ABB RAPID module: GoFa_GeneratedModule.modx

Module ACADIA_WORKSHOP_00_TEST
!Declarations

!jointtarget
VAR jointtarget TGofa_InitialConfig:=[[0,0,0,0,90,0],[9E9,9E9,9E9,9E9,9E9,9E9]];

!robtarget (Not Used for MoveAbsJ)
!VAR robtarget TGofa_0_End:=[[365,77.458,68.392],[0.707107,0,0,0.707107],[-1,0,0,0],[9E9,9E9,9E9,9E9,9E9,9E9]];

!speeddata (mm/s for the TCP, degrees/s for reorientation of the tool, mm/s for linear external axes, degrees/s for rotating external axes)
VAR speeddata speeddata0:=[200,80,5000,1000];

!tooldata (Not Used)
!PERS tooldata PonGoFa:=[True,[[-36.666,0.002,138.175],[0,0.92388,0,0.382683]],[0.001,[0,0,0.1],[1,0,0,0],0,0,0]];

!wobjdata (Not Used for MoveAbsJ)
!PERS wobjdata Root:=[False,True,"",[[0,0,0],[1,0,0,0]],[[0,0,0],[1,0,0,0]]];

!zonedata (Blend)
VAR zonedata DefaultBlend:=[False,1,0.1,1,0.1,1,0.1];
VAR zonedata FinePoint:=[True,1,0.1,1,0.1,1,0.1];

Proc Main()
  !Path Acceleration Limitation, units is m/s2, syntax: PathAccLim AccLim [\AccMax] DecelLim [\DecelMax]
  PathAccLim TRUE\AccMax:=10,TRUE\DecelMax:=10;

  !Move Absolute Joint MoveAbsJ [\Conc] ToJointPos [\ID] [\NoEOffs] Speed [\V] | [\T] Zone [\Z] [\Inpos] Tool [\WObj]
  !Move to Initial Config
  MoveAbsJ TGofa_InitialConfig,speeddata0,FinePoint,tool0;  TPWrite "Action 0 FreeMovement.";
  MoveAbsJ [[0.00,0.00,0.00,0.00,0.00,0.00],[9E9,9E9,9E9,9E9,9E9,9E9]],speeddata0,DefaultBlend,tool0;
  MoveAbsJ [[-0.73,0.32,0.53,0.48,-0.90,0.98],[9E9,9E9,9E9,9E9,9E9,9E9]],speeddata0,DefaultBlend,tool0;
  MoveAbsJ [[-1.45,0.64,1.05,0.95,-1.81,1.96],[9E9,9E9,9E9,9E9,9E9,9E9]],speeddata0,DefaultBlend,tool0;
  MoveAbsJ [[-2.18,0.96,1.58,1.43,-2.71,2.94],[9E9,9E9,9E9,9E9,9E9,9E9]],speeddata0,DefaultBlend,tool0;
  MoveAbsJ [[-2.90,1.28,2.11,1.91,-3.62,3.92],[9E9,9E9,9E9,9E9,9E9,9E9]],speeddata0,DefaultBlend,tool0;
  MoveAbsJ [[-3.63,1.60,2.64,2.39,-4.52,4.90],[9E9,9E9,9E9,9E9,9E9,9E9]],speeddata0,DefaultBlend,tool0;
  MoveAbsJ [[-4.35,1.92,3.16,2.86,-5.43,5.88],[9E9,9E9,9E9,9E9,9E9,9E9]],speeddata0,DefaultBlend,tool0;
  MoveAbsJ [[-5.08,2.24,3.69,3.34,-6.33,6.86],[9E9,9E9,9E9,9E9,9E9,9E9]],speeddata0,DefaultBlend,tool0;
  MoveAbsJ [[-5.81,2.56,4.22,3.82,-7.24,7.84],[9E9,9E9,9E9,9E9,9E9,9E9]],speeddata0,DefaultBlend,tool0;
  MoveAbsJ [[-6.53,2.88,4.74,4.29,-8.14,8.82],[9E9,9E9,9E9,9E9,9E9,9E9]],speeddata0,DefaultBlend,tool0;
  MoveAbsJ [[-7.26,3.20,5.27,4.77,-9.05,9.80],[9E9,9E9,9E9,9E9,9E9,9E9]],speeddata0,DefaultBlend,tool0;
  MoveAbsJ [[-7.98,3.52,5.80,5.25,-9.95,10.78],[9E9,9E9,9E9,9E9,9E9,9E9]],speeddata0,DefaultBlend,tool0;
  MoveAbsJ [[-8.71,3.84,6.33,5.72,-10.86,11.76],[9E9,9E9,9E9,9E9,9E9,9E9]],speeddata0,DefaultBlend,tool0;
  MoveAbsJ [[-9.44,4.15,6.85,6.20,-11.76,12.74],[9E9,9E9,9E9,9E9,9E9,9E9]],speeddata0,DefaultBlend,tool0;
  MoveAbsJ [[-10.16,4.47,7.38,6.68,-12.67,13.72],[9E9,9E9,9E9,9E9,9E9,9E9]],speeddata0,DefaultBlend,tool0;
  MoveAbsJ [[-10.89,4.79,7.91,7.16,-13.57,14.70],[9E9,9E9,9E9,9E9,9E9,9E9]],speeddata0,DefaultBlend,tool0;
  MoveAbsJ [[-11.61,5.11,8.43,7.63,-14.48,15.68],[9E9,9E9,9E9,9E9,9E9,9E9]],speeddata0,DefaultBlend,tool0;
  MoveAbsJ [[-12.34,5.43,8.96,8.11,-15.38,16.66],[9E9,9E9,9E9,9E9,9E9,9E9]],speeddata0,DefaultBlend,tool0;
  MoveAbsJ [[-13.06,5.75,9.49,8.59,-16.29,17.64],[9E9,9E9,9E9,9E9,9E9,9E9]],speeddata0,DefaultBlend,tool0;
  MoveAbsJ [[-13.79,6.07,10.02,9.06,-17.19,18.62],[9E9,9E9,9E9,9E9,9E9,9E9]],speeddata0,DefaultBlend,tool0;
  MoveAbsJ [[-14.52,6.39,10.54,9.54,-18.10,19.60],[9E9,9E9,9E9,9E9,9E9,9E9]],speeddata0,DefaultBlend,tool0;
  MoveAbsJ [[-15.24,6.71,11.07,10.02,-19.00,20.58],[9E9,9E9,9E9,9E9,9E9,9E9]],speeddata0,DefaultBlend,tool0;
  MoveAbsJ [[-15.97,7.03,11.60,10.50,-19.91,21.56],[9E9,9E9,9E9,9E9,9E9,9E9]],speeddata0,DefaultBlend,tool0;
  MoveAbsJ [[-16.69,7.35,12.12,10.97,-20.81,22.54],[9E9,9E9,9E9,9E9,9E9,9E9]],speeddata0,DefaultBlend,tool0;
  MoveAbsJ [[-17.42,7.67,12.65,11.45,-21.72,23.52],[9E9,9E9,9E9,9E9,9E9,9E9]],speeddata0,DefaultBlend,tool0;
  MoveAbsJ [[-18.15,7.99,13.18,11.93,-22.62,24.50],[9E9,9E9,9E9,9E9,9E9,9E9]],speeddata0,DefaultBlend,tool0;
  MoveAbsJ [[-18.87,8.31,13.71,12.40,-23.53,25.48],[9E9,9E9,9E9,9E9,9E9,9E9]],speeddata0,DefaultBlend,tool0;
  MoveAbsJ [[-19.60,8.63,14.23,12.88,-24.43,26.46],[9E9,9E9,9E9,9E9,9E9,9E9]],speeddata0,DefaultBlend,tool0;
  MoveAbsJ [[-20.32,8.95,14.76,13.36,-25.34,27.44],[9E9,9E9,9E9,9E9,9E9,9E9]],speeddata0,DefaultBlend,tool0;
  MoveAbsJ [[-21.05,9.27,15.29,13.84,-26.24,28.42],[9E9,9E9,9E9,9E9,9E9,9E9]],speeddata0,DefaultBlend,tool0;
  MoveAbsJ [[-21.77,9.59,15.81,14.31,-27.15,29.40],[9E9,9E9,9E9,9E9,9E9,9E9]],speeddata0,DefaultBlend,tool0;
  MoveAbsJ [[-22.50,9.91,16.34,14.79,-28.05,30.38],[9E9,9E9,9E9,9E9,9E9,9E9]],speeddata0,DefaultBlend,tool0;
  MoveAbsJ [[-23.23,10.23,16.87,15.27,-28.96,31.36],[9E9,9E9,9E9,9E9,9E9,9E9]],speeddata0,DefaultBlend,tool0;
  MoveAbsJ [[-23.95,10.55,17.40,15.74,-29.86,32.34],[9E9,9E9,9E9,9E9,9E9,9E9]],speeddata0,DefaultBlend,tool0;
  MoveAbsJ [[-24.68,10.87,17.92,16.22,-30.77,33.32],[9E9,9E9,9E9,9E9,9E9,9E9]],speeddata0,DefaultBlend,tool0;
  MoveAbsJ [[-25.40,11.19,18.45,16.70,-31.67,34.30],[9E9,9E9,9E9,9E9,9E9,9E9]],speeddata0,DefaultBlend,tool0;
  MoveAbsJ [[-26.13,11.51,18.98,17.17,-32.58,35.28],[9E9,9E9,9E9,9E9,9E9,9E9]],speeddata0,DefaultBlend,tool0;
  MoveAbsJ [[-26.85,11.83,19.50,17.65,-33.48,36.26],[9E9,9E9,9E9,9E9,9E9,9E9]],speeddata0,DefaultBlend,tool0;
  MoveAbsJ [[-27.58,12.15,20.03,18.13,-34.39,37.24],[9E9,9E9,9E9,9E9,9E9,9E9]],speeddata0,DefaultBlend,tool0;
  MoveAbsJ [[-28.31,12.46,20.56,18.61,-35.29,38.22],[9E9,9E9,9E9,9E9,9E9,9E9]],speeddata0,DefaultBlend,tool0;
  MoveAbsJ [[-29.03,12.78,21.09,19.08,-36.20,39.20],[9E9,9E9,9E9,9E9,9E9,9E9]],speeddata0,DefaultBlend,tool0;
  MoveAbsJ [[-29.76,13.10,21.61,19.56,-37.10,40.18],[9E9,9E9,9E9,9E9,9E9,9E9]],speeddata0,DefaultBlend,tool0;
  MoveAbsJ [[-30.48,13.42,22.14,20.04,-38.01,41.17],[9E9,9E9,9E9,9E9,9E9,9E9]],speeddata0,DefaultBlend,tool0;
  MoveAbsJ [[-31.21,13.74,22.67,20.51,-38.91,42.15],[9E9,9E9,9E9,9E9,9E9,9E9]],speeddata0,DefaultBlend,tool0;
  MoveAbsJ [[-31.94,14.06,23.19,20.99,-39.82,43.13],[9E9,9E9,9E9,9E9,9E9,9E9]],speeddata0,DefaultBlend,tool0;
  MoveAbsJ [[-32.66,14.38,23.72,21.47,-40.72,44.11],[9E9,9E9,9E9,9E9,9E9,9E9]],speeddata0,DefaultBlend,tool0;
  MoveAbsJ [[-33.39,14.70,24.25,21.95,-41.63,45.09],[9E9,9E9,9E9,9E9,9E9,9E9]],speeddata0,DefaultBlend,tool0;
  MoveAbsJ [[-34.11,15.02,24.78,22.42,-42.53,46.07],[9E9,9E9,9E9,9E9,9E9,9E9]],speeddata0,DefaultBlend,tool0;
  MoveAbsJ [[-34.84,15.34,25.30,22.90,-43.44,47.05],[9E9,9E9,9E9,9E9,9E9,9E9]],speeddata0,DefaultBlend,tool0;
  MoveAbsJ [[-35.56,15.66,25.83,23.38,-44.34,48.03],[9E9,9E9,9E9,9E9,9E9,9E9]],speeddata0,DefaultBlend,tool0;
  MoveAbsJ [[-36.29,15.98,26.36,23.85,-45.25,49.01],[9E9,9E9,9E9,9E9,9E9,9E9]],speeddata0,DefaultBlend,tool0;
  MoveAbsJ [[-37.02,16.30,26.88,24.33,-46.15,49.99],[9E9,9E9,9E9,9E9,9E9,9E9]],speeddata0,DefaultBlend,tool0;
  MoveAbsJ [[-37.74,16.62,27.41,24.81,-47.06,50.97],[9E9,9E9,9E9,9E9,9E9,9E9]],speeddata0,DefaultBlend,tool0;
  MoveAbsJ [[-38.47,16.94,27.94,25.29,-47.96,51.95],[9E9,9E9,9E9,9E9,9E9,9E9]],speeddata0,DefaultBlend,tool0;
  MoveAbsJ [[-39.19,17.26,28.47,25.76,-48.87,52.93],[9E9,9E9,9E9,9E9,9E9,9E9]],speeddata0,DefaultBlend,tool0;
  MoveAbsJ [[-39.92,17.58,28.99,26.24,-49.77,53.91],[9E9,9E9,9E9,9E9,9E9,9E9]],speeddata0,DefaultBlend,tool0;
  MoveAbsJ [[-40.64,17.90,29.52,26.72,-50.68,54.89],[9E9,9E9,9E9,9E9,9E9,9E9]],speeddata0,DefaultBlend,tool0;
  MoveAbsJ [[-41.37,18.22,30.05,27.19,-51.58,55.87],[9E9,9E9,9E9,9E9,9E9,9E9]],speeddata0,DefaultBlend,tool0;
  MoveAbsJ [[-42.10,18.54,30.57,27.67,-52.49,56.85],[9E9,9E9,9E9,9E9,9E9,9E9]],speeddata0,DefaultBlend,tool0;
  MoveAbsJ [[-42.82,18.86,31.10,28.15,-53.39,57.83],[9E9,9E9,9E9,9E9,9E9,9E9]],speeddata0,DefaultBlend,tool0;
  MoveAbsJ [[-43.55,19.18,31.63,28.62,-54.29,58.81],[9E9,9E9,9E9,9E9,9E9,9E9]],speeddata0,DefaultBlend,tool0;
  MoveAbsJ [[-44.27,19.50,32.16,29.10,-55.20,59.79],[9E9,9E9,9E9,9E9,9E9,9E9]],speeddata0,DefaultBlend,tool0;
  MoveAbsJ [[-45.00,19.82,32.68,29.58,-56.10,60.77],[9E9,9E9,9E9,9E9,9E9,9E9]],speeddata0,DefaultBlend,tool0;
  MoveAbsJ [[-45.73,20.14,33.21,30.06,-57.01,61.75],[9E9,9E9,9E9,9E9,9E9,9E9]],speeddata0,DefaultBlend,tool0;
  MoveAbsJ [[-46.45,20.46,33.74,30.53,-57.91,62.73],[9E9,9E9,9E9,9E9,9E9,9E9]],speeddata0,DefaultBlend,tool0;
  MoveAbsJ [[-47.18,20.77,34.26,31.01,-58.82,63.71],[9E9,9E9,9E9,9E9,9E9,9E9]],speeddata0,DefaultBlend,tool0;
  MoveAbsJ [[-47.90,21.09,34.79,31.49,-59.72,64.69],[9E9,9E9,9E9,9E9,9E9,9E9]],speeddata0,DefaultBlend,tool0;
  MoveAbsJ [[-48.63,21.41,35.32,31.96,-60.63,65.67],[9E9,9E9,9E9,9E9,9E9,9E9]],speeddata0,DefaultBlend,tool0;
  MoveAbsJ [[-49.35,21.73,35.85,32.44,-61.53,66.65],[9E9,9E9,9E9,9E9,9E9,9E9]],speeddata0,DefaultBlend,tool0;
  MoveAbsJ [[-50.08,22.05,36.37,32.92,-62.44,67.63],[9E9,9E9,9E9,9E9,9E9,9E9]],speeddata0,DefaultBlend,tool0;
  MoveAbsJ [[-50.81,22.37,36.90,33.40,-63.34,68.61],[9E9,9E9,9E9,9E9,9E9,9E9]],speeddata0,DefaultBlend,tool0;
  MoveAbsJ [[-51.53,22.69,37.43,33.87,-64.25,69.59],[9E9,9E9,9E9,9E9,9E9,9E9]],speeddata0,DefaultBlend,tool0;
  MoveAbsJ [[-52.26,23.01,37.95,34.35,-65.15,70.57],[9E9,9E9,9E9,9E9,9E9,9E9]],speeddata0,DefaultBlend,tool0;
  MoveAbsJ [[-52.98,23.33,38.48,34.83,-66.06,71.55],[9E9,9E9,9E9,9E9,9E9,9E9]],speeddata0,DefaultBlend,tool0;
  MoveAbsJ [[-53.71,23.65,39.01,35.30,-66.96,72.53],[9E9,9E9,9E9,9E9,9E9,9E9]],speeddata0,DefaultBlend,tool0;
  MoveAbsJ [[-54.44,23.97,39.54,35.78,-67.87,73.51],[9E9,9E9,9E9,9E9,9E9,9E9]],speeddata0,DefaultBlend,tool0;
  MoveAbsJ [[-55.16,24.29,40.06,36.26,-68.77,74.49],[9E9,9E9,9E9,9E9,9E9,9E9]],speeddata0,DefaultBlend,tool0;
  MoveAbsJ [[-55.89,24.61,40.59,36.74,-69.68,75.47],[9E9,9E9,9E9,9E9,9E9,9E9]],speeddata0,FinePoint,tool0;
  TPWrite "Action 1 LoadWorkpiece.";
  TPWrite "Press Play to Continue";
  Stop;
  TPWrite "Action 2 CloseGripper.";
  TPWrite "Press Play to Continue";
  Stop;
  TPWrite "Action 3 FreeMovement.";
  MoveAbsJ [[-55.89,24.61,40.59,36.74,-69.68,75.47],[9E9,9E9,9E9,9E9,9E9,9E9]],speeddata0,DefaultBlend,tool0;
  MoveAbsJ [[-55.58,24.66,40.49,36.58,-69.24,74.48],[9E9,9E9,9E9,9E9,9E9,9E9]],speeddata0,DefaultBlend,tool0;
  MoveAbsJ [[-55.26,24.72,40.40,36.43,-68.80,73.49],[9E9,9E9,9E9,9E9,9E9,9E9]],speeddata0,DefaultBlend,tool0;
  MoveAbsJ [[-54.95,24.77,40.30,36.27,-68.36,72.49],[9E9,9E9,9E9,9E9,9E9,9E9]],speeddata0,DefaultBlend,tool0;
  MoveAbsJ [[-54.64,24.82,40.20,36.12,-67.92,71.50],[9E9,9E9,9E9,9E9,9E9,9E9]],speeddata0,DefaultBlend,tool0;
  MoveAbsJ [[-54.33,24.87,40.10,35.97,-67.48,70.51],[9E9,9E9,9E9,9E9,9E9,9E9]],speeddata0,DefaultBlend,tool0;
  MoveAbsJ [[-54.02,24.93,40.00,35.81,-67.03,69.52],[9E9,9E9,9E9,9E9,9E9,9E9]],speeddata0,DefaultBlend,tool0;
  MoveAbsJ [[-53.71,24.98,39.91,35.66,-66.59,68.53],[9E9,9E9,9E9,9E9,9E9,9E9]],speeddata0,DefaultBlend,tool0;
  MoveAbsJ [[-53.40,25.03,39.81,35.51,-66.15,67.53],[9E9,9E9,9E9,9E9,9E9,9E9]],speeddata0,DefaultBlend,tool0;
  MoveAbsJ [[-53.09,25.08,39.71,35.35,-65.71,66.54],[9E9,9E9,9E9,9E9,9E9,9E9]],speeddata0,DefaultBlend,tool0;
  MoveAbsJ [[-52.78,25.14,39.61,35.20,-65.27,65.55],[9E9,9E9,9E9,9E9,9E9,9E9]],speeddata0,DefaultBlend,tool0;
  MoveAbsJ [[-52.47,25.19,39.51,35.04,-64.83,64.56],[9E9,9E9,9E9,9E9,9E9,9E9]],speeddata0,DefaultBlend,tool0;
  MoveAbsJ [[-52.16,25.24,39.42,34.89,-64.39,63.57],[9E9,9E9,9E9,9E9,9E9,9E9]],speeddata0,DefaultBlend,tool0;
  MoveAbsJ [[-51.84,25.29,39.32,34.74,-63.95,62.58],[9E9,9E9,9E9,9E9,9E9,9E9]],speeddata0,DefaultBlend,tool0;
  MoveAbsJ [[-51.53,25.35,39.22,34.58,-63.51,61.58],[9E9,9E9,9E9,9E9,9E9,9E9]],speeddata0,DefaultBlend,tool0;
  MoveAbsJ [[-51.22,25.40,39.12,34.43,-63.07,60.59],[9E9,9E9,9E9,9E9,9E9,9E9]],speeddata0,DefaultBlend,tool0;
  MoveAbsJ [[-50.91,25.45,39.03,34.28,-62.63,59.60],[9E9,9E9,9E9,9E9,9E9,9E9]],speeddata0,DefaultBlend,tool0;
  MoveAbsJ [[-50.60,25.50,38.93,34.12,-62.19,58.61],[9E9,9E9,9E9,9E9,9E9,9E9]],speeddata0,DefaultBlend,tool0;
  MoveAbsJ [[-50.29,25.56,38.83,33.97,-61.75,57.62],[9E9,9E9,9E9,9E9,9E9,9E9]],speeddata0,DefaultBlend,tool0;
  MoveAbsJ [[-49.98,25.61,38.73,33.81,-61.31,56.63],[9E9,9E9,9E9,9E9,9E9,9E9]],speeddata0,DefaultBlend,tool0;
  MoveAbsJ [[-49.67,25.66,38.63,33.66,-60.87,55.63],[9E9,9E9,9E9,9E9,9E9,9E9]],speeddata0,DefaultBlend,tool0;
  MoveAbsJ [[-49.36,25.71,38.54,33.51,-60.42,54.64],[9E9,9E9,9E9,9E9,9E9,9E9]],speeddata0,DefaultBlend,tool0;
  MoveAbsJ [[-49.05,25.77,38.44,33.35,-59.98,53.65],[9E9,9E9,9E9,9E9,9E9,9E9]],speeddata0,DefaultBlend,tool0;
  MoveAbsJ [[-48.73,25.82,38.34,33.20,-59.54,52.66],[9E9,9E9,9E9,9E9,9E9,9E9]],speeddata0,DefaultBlend,tool0;
  MoveAbsJ [[-48.42,25.87,38.24,33.05,-59.10,51.67],[9E9,9E9,9E9,9E9,9E9,9E9]],speeddata0,DefaultBlend,tool0;
  MoveAbsJ [[-48.11,25.92,38.14,32.89,-58.66,50.67],[9E9,9E9,9E9,9E9,9E9,9E9]],speeddata0,DefaultBlend,tool0;
  MoveAbsJ [[-47.80,25.98,38.05,32.74,-58.22,49.68],[9E9,9E9,9E9,9E9,9E9,9E9]],speeddata0,DefaultBlend,tool0;
  MoveAbsJ [[-47.49,26.03,37.95,32.59,-57.78,48.69],[9E9,9E9,9E9,9E9,9E9,9E9]],speeddata0,DefaultBlend,tool0;
  MoveAbsJ [[-47.18,26.08,37.85,32.43,-57.34,47.70],[9E9,9E9,9E9,9E9,9E9,9E9]],speeddata0,DefaultBlend,tool0;
  MoveAbsJ [[-46.87,26.13,37.75,32.28,-56.90,46.71],[9E9,9E9,9E9,9E9,9E9,9E9]],speeddata0,DefaultBlend,tool0;
  MoveAbsJ [[-46.56,26.18,37.66,32.12,-56.46,45.72],[9E9,9E9,9E9,9E9,9E9,9E9]],speeddata0,DefaultBlend,tool0;
  MoveAbsJ [[-46.25,26.24,37.56,31.97,-56.02,44.72],[9E9,9E9,9E9,9E9,9E9,9E9]],speeddata0,DefaultBlend,tool0;
  MoveAbsJ [[-45.94,26.29,37.46,31.82,-55.58,43.73],[9E9,9E9,9E9,9E9,9E9,9E9]],speeddata0,DefaultBlend,tool0;
  MoveAbsJ [[-45.62,26.34,37.36,31.66,-55.14,42.74],[9E9,9E9,9E9,9E9,9E9,9E9]],speeddata0,DefaultBlend,tool0;
  MoveAbsJ [[-45.31,26.39,37.26,31.51,-54.70,41.75],[9E9,9E9,9E9,9E9,9E9,9E9]],speeddata0,DefaultBlend,tool0;
  MoveAbsJ [[-45.00,26.45,37.17,31.36,-54.26,40.76],[9E9,9E9,9E9,9E9,9E9,9E9]],speeddata0,DefaultBlend,tool0;
  MoveAbsJ [[-44.69,26.50,37.07,31.20,-53.81,39.77],[9E9,9E9,9E9,9E9,9E9,9E9]],speeddata0,DefaultBlend,tool0;
  MoveAbsJ [[-44.38,26.55,36.97,31.05,-53.37,38.77],[9E9,9E9,9E9,9E9,9E9,9E9]],speeddata0,DefaultBlend,tool0;
  MoveAbsJ [[-44.07,26.60,36.87,30.89,-52.93,37.78],[9E9,9E9,9E9,9E9,9E9,9E9]],speeddata0,DefaultBlend,tool0;
  MoveAbsJ [[-43.76,26.66,36.77,30.74,-52.49,36.79],[9E9,9E9,9E9,9E9,9E9,9E9]],speeddata0,DefaultBlend,tool0;
  MoveAbsJ [[-43.45,26.71,36.68,30.59,-52.05,35.80],[9E9,9E9,9E9,9E9,9E9,9E9]],speeddata0,DefaultBlend,tool0;
  MoveAbsJ [[-43.14,26.76,36.58,30.43,-51.61,34.81],[9E9,9E9,9E9,9E9,9E9,9E9]],speeddata0,DefaultBlend,tool0;
  MoveAbsJ [[-42.83,26.81,36.48,30.28,-51.17,33.81],[9E9,9E9,9E9,9E9,9E9,9E9]],speeddata0,DefaultBlend,tool0;
  MoveAbsJ [[-42.52,26.87,36.38,30.13,-50.73,32.82],[9E9,9E9,9E9,9E9,9E9,9E9]],speeddata0,DefaultBlend,tool0;
  MoveAbsJ [[-42.20,26.92,36.29,29.97,-50.29,31.83],[9E9,9E9,9E9,9E9,9E9,9E9]],speeddata0,DefaultBlend,tool0;
  MoveAbsJ [[-41.89,26.97,36.19,29.82,-49.85,30.84],[9E9,9E9,9E9,9E9,9E9,9E9]],speeddata0,DefaultBlend,tool0;
  MoveAbsJ [[-41.58,27.02,36.09,29.66,-49.41,29.85],[9E9,9E9,9E9,9E9,9E9,9E9]],speeddata0,DefaultBlend,tool0;
  MoveAbsJ [[-41.27,27.08,35.99,29.51,-48.97,28.86],[9E9,9E9,9E9,9E9,9E9,9E9]],speeddata0,DefaultBlend,tool0;
  MoveAbsJ [[-40.96,27.13,35.89,29.36,-48.53,27.86],[9E9,9E9,9E9,9E9,9E9,9E9]],speeddata0,DefaultBlend,tool0;
  MoveAbsJ [[-40.65,27.18,35.80,29.20,-48.09,26.87],[9E9,9E9,9E9,9E9,9E9,9E9]],speeddata0,DefaultBlend,tool0;
  MoveAbsJ [[-40.34,27.23,35.70,29.05,-47.65,25.88],[9E9,9E9,9E9,9E9,9E9,9E9]],speeddata0,DefaultBlend,tool0;
  MoveAbsJ [[-40.03,27.29,35.60,28.90,-47.21,24.89],[9E9,9E9,9E9,9E9,9E9,9E9]],speeddata0,DefaultBlend,tool0;
  MoveAbsJ [[-39.72,27.34,35.50,28.74,-46.76,23.90],[9E9,9E9,9E9,9E9,9E9,9E9]],speeddata0,DefaultBlend,tool0;
  MoveAbsJ [[-39.41,27.39,35.40,28.59,-46.32,22.91],[9E9,9E9,9E9,9E9,9E9,9E9]],speeddata0,DefaultBlend,tool0;
  MoveAbsJ [[-39.09,27.44,35.31,28.44,-45.88,21.91],[9E9,9E9,9E9,9E9,9E9,9E9]],speeddata0,DefaultBlend,tool0;
  MoveAbsJ [[-38.78,27.50,35.21,28.28,-45.44,20.92],[9E9,9E9,9E9,9E9,9E9,9E9]],speeddata0,DefaultBlend,tool0;
  MoveAbsJ [[-38.47,27.55,35.11,28.13,-45.00,19.93],[9E9,9E9,9E9,9E9,9E9,9E9]],speeddata0,DefaultBlend,tool0;
  MoveAbsJ [[-38.16,27.60,35.01,27.97,-44.56,18.94],[9E9,9E9,9E9,9E9,9E9,9E9]],speeddata0,DefaultBlend,tool0;
  MoveAbsJ [[-37.85,27.65,34.92,27.82,-44.12,17.95],[9E9,9E9,9E9,9E9,9E9,9E9]],speeddata0,DefaultBlend,tool0;
  MoveAbsJ [[-37.54,27.71,34.82,27.67,-43.68,16.95],[9E9,9E9,9E9,9E9,9E9,9E9]],speeddata0,DefaultBlend,tool0;
  MoveAbsJ [[-37.23,27.76,34.72,27.51,-43.24,15.96],[9E9,9E9,9E9,9E9,9E9,9E9]],speeddata0,DefaultBlend,tool0;
  MoveAbsJ [[-36.92,27.81,34.62,27.36,-42.80,14.97],[9E9,9E9,9E9,9E9,9E9,9E9]],speeddata0,DefaultBlend,tool0;
  MoveAbsJ [[-36.61,27.86,34.52,27.21,-42.36,13.98],[9E9,9E9,9E9,9E9,9E9,9E9]],speeddata0,DefaultBlend,tool0;
  MoveAbsJ [[-36.30,27.92,34.43,27.05,-41.92,12.99],[9E9,9E9,9E9,9E9,9E9,9E9]],speeddata0,DefaultBlend,tool0;
  MoveAbsJ [[-35.98,27.97,34.33,26.90,-41.48,12.00],[9E9,9E9,9E9,9E9,9E9,9E9]],speeddata0,DefaultBlend,tool0;
  MoveAbsJ [[-35.67,28.02,34.23,26.74,-41.04,11.00],[9E9,9E9,9E9,9E9,9E9,9E9]],speeddata0,DefaultBlend,tool0;
  MoveAbsJ [[-35.36,28.07,34.13,26.59,-40.60,10.01],[9E9,9E9,9E9,9E9,9E9,9E9]],speeddata0,DefaultBlend,tool0;
  MoveAbsJ [[-35.05,28.13,34.03,26.44,-40.15,9.02],[9E9,9E9,9E9,9E9,9E9,9E9]],speeddata0,DefaultBlend,tool0;
  MoveAbsJ [[-34.74,28.18,33.94,26.28,-39.71,8.03],[9E9,9E9,9E9,9E9,9E9,9E9]],speeddata0,DefaultBlend,tool0;
  MoveAbsJ [[-34.43,28.23,33.84,26.13,-39.27,7.04],[9E9,9E9,9E9,9E9,9E9,9E9]],speeddata0,DefaultBlend,tool0;
  MoveAbsJ [[-34.12,28.28,33.74,25.98,-38.83,6.04],[9E9,9E9,9E9,9E9,9E9,9E9]],speeddata0,DefaultBlend,tool0;
  MoveAbsJ [[-33.81,28.34,33.64,25.82,-38.39,5.05],[9E9,9E9,9E9,9E9,9E9,9E9]],speeddata0,DefaultBlend,tool0;
  MoveAbsJ [[-33.50,28.39,33.55,25.67,-37.95,4.06],[9E9,9E9,9E9,9E9,9E9,9E9]],speeddata0,DefaultBlend,tool0;
  MoveAbsJ [[-33.19,28.44,33.45,25.51,-37.51,3.07],[9E9,9E9,9E9,9E9,9E9,9E9]],speeddata0,DefaultBlend,tool0;
  MoveAbsJ [[-32.88,28.49,33.35,25.36,-37.07,2.08],[9E9,9E9,9E9,9E9,9E9,9E9]],speeddata0,DefaultBlend,tool0;
  MoveAbsJ [[-32.56,28.55,33.25,25.21,-36.63,1.09],[9E9,9E9,9E9,9E9,9E9,9E9]],speeddata0,DefaultBlend,tool0;
  MoveAbsJ [[-32.25,28.60,33.15,25.05,-36.19,0.09],[9E9,9E9,9E9,9E9,9E9,9E9]],speeddata0,DefaultBlend,tool0;
  MoveAbsJ [[-31.94,28.65,33.06,24.90,-35.75,-0.90],[9E9,9E9,9E9,9E9,9E9,9E9]],speeddata0,DefaultBlend,tool0;
  MoveAbsJ [[-31.63,28.70,32.96,24.75,-35.31,-1.89],[9E9,9E9,9E9,9E9,9E9,9E9]],speeddata0,DefaultBlend,tool0;
  MoveAbsJ [[-31.32,28.76,32.86,24.59,-34.87,-2.88],[9E9,9E9,9E9,9E9,9E9,9E9]],speeddata0,DefaultBlend,tool0;
  MoveAbsJ [[-31.01,28.81,32.76,24.44,-34.43,-3.87],[9E9,9E9,9E9,9E9,9E9,9E9]],speeddata0,DefaultBlend,tool0;
  MoveAbsJ [[-30.70,28.86,32.67,24.29,-33.99,-4.86],[9E9,9E9,9E9,9E9,9E9,9E9]],speeddata0,DefaultBlend,tool0;
  MoveAbsJ [[-30.39,28.91,32.57,24.13,-33.54,-5.86],[9E9,9E9,9E9,9E9,9E9,9E9]],speeddata0,DefaultBlend,tool0;
  MoveAbsJ [[-30.08,28.97,32.47,23.98,-33.10,-6.85],[9E9,9E9,9E9,9E9,9E9,9E9]],speeddata0,DefaultBlend,tool0;
  MoveAbsJ [[-29.77,29.02,32.37,23.82,-32.66,-7.84],[9E9,9E9,9E9,9E9,9E9,9E9]],speeddata0,DefaultBlend,tool0;
  MoveAbsJ [[-29.45,29.07,32.27,23.67,-32.22,-8.83],[9E9,9E9,9E9,9E9,9E9,9E9]],speeddata0,DefaultBlend,tool0;
  MoveAbsJ [[-29.14,29.12,32.18,23.52,-31.78,-9.82],[9E9,9E9,9E9,9E9,9E9,9E9]],speeddata0,DefaultBlend,tool0;
  MoveAbsJ [[-28.83,29.18,32.08,23.36,-31.34,-10.82],[9E9,9E9,9E9,9E9,9E9,9E9]],speeddata0,DefaultBlend,tool0;
  MoveAbsJ [[-28.52,29.23,31.98,23.21,-30.90,-11.81],[9E9,9E9,9E9,9E9,9E9,9E9]],speeddata0,DefaultBlend,tool0;
  MoveAbsJ [[-28.21,29.28,31.88,23.06,-30.46,-12.80],[9E9,9E9,9E9,9E9,9E9,9E9]],speeddata0,DefaultBlend,tool0;
  MoveAbsJ [[-27.90,29.33,31.78,22.90,-30.02,-13.79],[9E9,9E9,9E9,9E9,9E9,9E9]],speeddata0,DefaultBlend,tool0;
  MoveAbsJ [[-27.59,29.39,31.69,22.75,-29.58,-14.78],[9E9,9E9,9E9,9E9,9E9,9E9]],speeddata0,DefaultBlend,tool0;
  MoveAbsJ [[-27.28,29.44,31.59,22.59,-29.14,-15.77],[9E9,9E9,9E9,9E9,9E9,9E9]],speeddata0,DefaultBlend,tool0;
  MoveAbsJ [[-26.97,29.49,31.49,22.44,-28.70,-16.77],[9E9,9E9,9E9,9E9,9E9,9E9]],speeddata0,DefaultBlend,tool0;
  MoveAbsJ [[-26.66,29.54,31.39,22.29,-28.26,-17.76],[9E9,9E9,9E9,9E9,9E9,9E9]],speeddata0,DefaultBlend,tool0;
  MoveAbsJ [[-26.34,29.60,31.30,22.13,-27.82,-18.75],[9E9,9E9,9E9,9E9,9E9,9E9]],speeddata0,DefaultBlend,tool0;
  MoveAbsJ [[-26.03,29.65,31.20,21.98,-27.38,-19.74],[9E9,9E9,9E9,9E9,9E9,9E9]],speeddata0,DefaultBlend,tool0;
  MoveAbsJ [[-25.72,29.70,31.10,21.83,-26.93,-20.73],[9E9,9E9,9E9,9E9,9E9,9E9]],speeddata0,DefaultBlend,tool0;
  MoveAbsJ [[-25.41,29.75,31.00,21.67,-26.49,-21.72],[9E9,9E9,9E9,9E9,9E9,9E9]],speeddata0,DefaultBlend,tool0;
  MoveAbsJ [[-25.10,29.81,30.90,21.52,-26.05,-22.72],[9E9,9E9,9E9,9E9,9E9,9E9]],speeddata0,DefaultBlend,tool0;
  MoveAbsJ [[-24.79,29.86,30.81,21.36,-25.61,-23.71],[9E9,9E9,9E9,9E9,9E9,9E9]],speeddata0,DefaultBlend,tool0;
  MoveAbsJ [[-24.48,29.91,30.71,21.21,-25.17,-24.70],[9E9,9E9,9E9,9E9,9E9,9E9]],speeddata0,DefaultBlend,tool0;
  MoveAbsJ [[-24.17,29.96,30.61,21.06,-24.73,-25.69],[9E9,9E9,9E9,9E9,9E9,9E9]],speeddata0,DefaultBlend,tool0;
  MoveAbsJ [[-23.86,30.02,30.51,20.90,-24.29,-26.68],[9E9,9E9,9E9,9E9,9E9,9E9]],speeddata0,DefaultBlend,tool0;
  MoveAbsJ [[-23.55,30.07,30.41,20.75,-23.85,-27.68],[9E9,9E9,9E9,9E9,9E9,9E9]],speeddata0,DefaultBlend,tool0;
  MoveAbsJ [[-23.23,30.12,30.32,20.60,-23.41,-28.67],[9E9,9E9,9E9,9E9,9E9,9E9]],speeddata0,DefaultBlend,tool0;
  MoveAbsJ [[-22.92,30.17,30.22,20.44,-22.97,-29.66],[9E9,9E9,9E9,9E9,9E9,9E9]],speeddata0,DefaultBlend,tool0;
  MoveAbsJ [[-22.61,30.23,30.12,20.29,-22.53,-30.65],[9E9,9E9,9E9,9E9,9E9,9E9]],speeddata0,DefaultBlend,tool0;
  MoveAbsJ [[-22.30,30.28,30.02,20.14,-22.09,-31.64],[9E9,9E9,9E9,9E9,9E9,9E9]],speeddata0,DefaultBlend,tool0;
  MoveAbsJ [[-21.99,30.33,29.93,19.98,-21.65,-32.63],[9E9,9E9,9E9,9E9,9E9,9E9]],speeddata0,DefaultBlend,tool0;
  MoveAbsJ [[-21.68,30.38,29.83,19.83,-21.21,-33.63],[9E9,9E9,9E9,9E9,9E9,9E9]],speeddata0,DefaultBlend,tool0;
  MoveAbsJ [[-21.37,30.44,29.73,19.67,-20.77,-34.62],[9E9,9E9,9E9,9E9,9E9,9E9]],speeddata0,DefaultBlend,tool0;
  MoveAbsJ [[-21.06,30.49,29.63,19.52,-20.33,-35.61],[9E9,9E9,9E9,9E9,9E9,9E9]],speeddata0,DefaultBlend,tool0;
  MoveAbsJ [[-20.75,30.54,29.53,19.37,-19.88,-36.60],[9E9,9E9,9E9,9E9,9E9,9E9]],speeddata0,DefaultBlend,tool0;
  MoveAbsJ [[-20.44,30.59,29.44,19.21,-19.44,-37.59],[9E9,9E9,9E9,9E9,9E9,9E9]],speeddata0,DefaultBlend,tool0;
  MoveAbsJ [[-20.13,30.65,29.34,19.06,-19.00,-38.58],[9E9,9E9,9E9,9E9,9E9,9E9]],speeddata0,DefaultBlend,tool0;
  MoveAbsJ [[-19.81,30.70,29.24,18.91,-18.56,-39.58],[9E9,9E9,9E9,9E9,9E9,9E9]],speeddata0,DefaultBlend,tool0;
  MoveAbsJ [[-19.50,30.75,29.14,18.75,-18.12,-40.57],[9E9,9E9,9E9,9E9,9E9,9E9]],speeddata0,DefaultBlend,tool0;
  MoveAbsJ [[-19.19,30.80,29.04,18.60,-17.68,-41.56],[9E9,9E9,9E9,9E9,9E9,9E9]],speeddata0,DefaultBlend,tool0;
  MoveAbsJ [[-18.88,30.86,28.95,18.44,-17.24,-42.55],[9E9,9E9,9E9,9E9,9E9,9E9]],speeddata0,DefaultBlend,tool0;
  MoveAbsJ [[-18.57,30.91,28.85,18.29,-16.80,-43.54],[9E9,9E9,9E9,9E9,9E9,9E9]],speeddata0,DefaultBlend,tool0;
  MoveAbsJ [[-18.26,30.96,28.75,18.14,-16.36,-44.54],[9E9,9E9,9E9,9E9,9E9,9E9]],speeddata0,DefaultBlend,tool0;
  MoveAbsJ [[-17.95,31.01,28.65,17.98,-15.92,-45.53],[9E9,9E9,9E9,9E9,9E9,9E9]],speeddata0,DefaultBlend,tool0;
  MoveAbsJ [[-17.64,31.07,28.56,17.83,-15.48,-46.52],[9E9,9E9,9E9,9E9,9E9,9E9]],speeddata0,DefaultBlend,tool0;
  MoveAbsJ [[-17.33,31.12,28.46,17.68,-15.04,-47.51],[9E9,9E9,9E9,9E9,9E9,9E9]],speeddata0,DefaultBlend,tool0;
  MoveAbsJ [[-17.02,31.17,28.36,17.52,-14.60,-48.50],[9E9,9E9,9E9,9E9,9E9,9E9]],speeddata0,DefaultBlend,tool0;
  MoveAbsJ [[-16.70,31.22,28.26,17.37,-14.16,-49.49],[9E9,9E9,9E9,9E9,9E9,9E9]],speeddata0,DefaultBlend,tool0;
  MoveAbsJ [[-16.39,31.28,28.16,17.21,-13.72,-50.49],[9E9,9E9,9E9,9E9,9E9,9E9]],speeddata0,DefaultBlend,tool0;
  MoveAbsJ [[-16.08,31.33,28.07,17.06,-13.27,-51.48],[9E9,9E9,9E9,9E9,9E9,9E9]],speeddata0,DefaultBlend,tool0;
  MoveAbsJ [[-15.77,31.38,27.97,16.91,-12.83,-52.47],[9E9,9E9,9E9,9E9,9E9,9E9]],speeddata0,DefaultBlend,tool0;
  MoveAbsJ [[-15.46,31.43,27.87,16.75,-12.39,-53.46],[9E9,9E9,9E9,9E9,9E9,9E9]],speeddata0,DefaultBlend,tool0;
  MoveAbsJ [[-15.15,31.49,27.77,16.60,-11.95,-54.45],[9E9,9E9,9E9,9E9,9E9,9E9]],speeddata0,DefaultBlend,tool0;
  MoveAbsJ [[-14.84,31.54,27.67,16.45,-11.51,-55.45],[9E9,9E9,9E9,9E9,9E9,9E9]],speeddata0,DefaultBlend,tool0;
  MoveAbsJ [[-14.53,31.59,27.58,16.29,-11.07,-56.44],[9E9,9E9,9E9,9E9,9E9,9E9]],speeddata0,DefaultBlend,tool0;
  MoveAbsJ [[-14.22,31.64,27.48,16.14,-10.63,-57.43],[9E9,9E9,9E9,9E9,9E9,9E9]],speeddata0,DefaultBlend,tool0;
  MoveAbsJ [[-13.91,31.70,27.38,15.99,-10.19,-58.42],[9E9,9E9,9E9,9E9,9E9,9E9]],speeddata0,DefaultBlend,tool0;
  MoveAbsJ [[-13.59,31.75,27.28,15.83,-9.75,-59.41],[9E9,9E9,9E9,9E9,9E9,9E9]],speeddata0,DefaultBlend,tool0;
  MoveAbsJ [[-13.28,31.80,27.19,15.68,-9.31,-60.40],[9E9,9E9,9E9,9E9,9E9,9E9]],speeddata0,DefaultBlend,tool0;
  MoveAbsJ [[-12.97,31.85,27.09,15.52,-8.87,-61.40],[9E9,9E9,9E9,9E9,9E9,9E9]],speeddata0,DefaultBlend,tool0;
  MoveAbsJ [[-12.66,31.91,26.99,15.37,-8.43,-62.39],[9E9,9E9,9E9,9E9,9E9,9E9]],speeddata0,DefaultBlend,tool0;
  MoveAbsJ [[-12.35,31.96,26.89,15.22,-7.99,-63.38],[9E9,9E9,9E9,9E9,9E9,9E9]],speeddata0,DefaultBlend,tool0;
  MoveAbsJ [[-12.04,32.01,26.79,15.06,-7.55,-64.37],[9E9,9E9,9E9,9E9,9E9,9E9]],speeddata0,DefaultBlend,tool0;
  MoveAbsJ [[-11.73,32.06,26.70,14.91,-7.11,-65.36],[9E9,9E9,9E9,9E9,9E9,9E9]],speeddata0,DefaultBlend,tool0;
  MoveAbsJ [[-11.42,32.12,26.60,14.76,-6.66,-66.35],[9E9,9E9,9E9,9E9,9E9,9E9]],speeddata0,DefaultBlend,tool0;
  MoveAbsJ [[-11.11,32.17,26.50,14.60,-6.22,-67.35],[9E9,9E9,9E9,9E9,9E9,9E9]],speeddata0,DefaultBlend,tool0;
  MoveAbsJ [[-10.80,32.22,26.40,14.45,-5.78,-68.34],[9E9,9E9,9E9,9E9,9E9,9E9]],speeddata0,DefaultBlend,tool0;
  MoveAbsJ [[-10.49,32.27,26.31,14.29,-5.34,-69.33],[9E9,9E9,9E9,9E9,9E9,9E9]],speeddata0,DefaultBlend,tool0;
  MoveAbsJ [[-10.17,32.33,26.21,14.14,-4.90,-70.32],[9E9,9E9,9E9,9E9,9E9,9E9]],speeddata0,DefaultBlend,tool0;
  MoveAbsJ [[-9.86,32.38,26.11,13.99,-4.46,-71.31],[9E9,9E9,9E9,9E9,9E9,9E9]],speeddata0,DefaultBlend,tool0;
  MoveAbsJ [[-9.55,32.43,26.01,13.83,-4.02,-72.31],[9E9,9E9,9E9,9E9,9E9,9E9]],speeddata0,DefaultBlend,tool0;
  MoveAbsJ [[-9.24,32.48,25.91,13.68,-3.58,-73.30],[9E9,9E9,9E9,9E9,9E9,9E9]],speeddata0,DefaultBlend,tool0;
  MoveAbsJ [[-8.93,32.54,25.82,13.53,-3.14,-74.29],[9E9,9E9,9E9,9E9,9E9,9E9]],speeddata0,DefaultBlend,tool0;
  MoveAbsJ [[-8.62,32.59,25.72,13.37,-2.70,-75.28],[9E9,9E9,9E9,9E9,9E9,9E9]],speeddata0,DefaultBlend,tool0;
  MoveAbsJ [[-8.31,32.64,25.62,13.22,-2.26,-76.27],[9E9,9E9,9E9,9E9,9E9,9E9]],speeddata0,DefaultBlend,tool0;
  MoveAbsJ [[-8.00,32.69,25.52,13.06,-1.82,-77.26],[9E9,9E9,9E9,9E9,9E9,9E9]],speeddata0,DefaultBlend,tool0;
  MoveAbsJ [[-7.69,32.75,25.42,12.91,-1.38,-78.26],[9E9,9E9,9E9,9E9,9E9,9E9]],speeddata0,DefaultBlend,tool0;
  MoveAbsJ [[-7.38,32.80,25.33,12.76,-0.94,-79.25],[9E9,9E9,9E9,9E9,9E9,9E9]],speeddata0,DefaultBlend,tool0;
  MoveAbsJ [[-7.06,32.85,25.23,12.60,-0.50,-80.24],[9E9,9E9,9E9,9E9,9E9,9E9]],speeddata0,DefaultBlend,tool0;
  MoveAbsJ [[-6.75,32.90,25.13,12.45,-0.05,-81.23],[9E9,9E9,9E9,9E9,9E9,9E9]],speeddata0,DefaultBlend,tool0;
  MoveAbsJ [[-6.44,32.96,25.03,12.30,0.39,-82.22],[9E9,9E9,9E9,9E9,9E9,9E9]],speeddata0,DefaultBlend,tool0;
  MoveAbsJ [[-6.13,33.01,24.94,12.14,0.83,-83.21],[9E9,9E9,9E9,9E9,9E9,9E9]],speeddata0,DefaultBlend,tool0;
  MoveAbsJ [[-5.82,33.06,24.84,11.99,1.27,-84.21],[9E9,9E9,9E9,9E9,9E9,9E9]],speeddata0,DefaultBlend,tool0;
  MoveAbsJ [[-5.51,33.11,24.74,11.84,1.71,-85.20],[9E9,9E9,9E9,9E9,9E9,9E9]],speeddata0,DefaultBlend,tool0;
  MoveAbsJ [[-5.20,33.17,24.64,11.68,2.15,-86.19],[9E9,9E9,9E9,9E9,9E9,9E9]],speeddata0,DefaultBlend,tool0;
  MoveAbsJ [[-4.89,33.22,24.54,11.53,2.59,-87.18],[9E9,9E9,9E9,9E9,9E9,9E9]],speeddata0,DefaultBlend,tool0;
  MoveAbsJ [[-4.58,33.27,24.45,11.37,3.03,-88.17],[9E9,9E9,9E9,9E9,9E9,9E9]],speeddata0,DefaultBlend,tool0;
  MoveAbsJ [[-4.27,33.32,24.35,11.22,3.47,-89.17],[9E9,9E9,9E9,9E9,9E9,9E9]],speeddata0,DefaultBlend,tool0;
  MoveAbsJ [[-3.95,33.38,24.25,11.07,3.91,-90.16],[9E9,9E9,9E9,9E9,9E9,9E9]],speeddata0,DefaultBlend,tool0;
  MoveAbsJ [[-3.64,33.43,24.15,10.91,4.35,-91.15],[9E9,9E9,9E9,9E9,9E9,9E9]],speeddata0,DefaultBlend,tool0;
  MoveAbsJ [[-3.33,33.48,24.05,10.76,4.79,-92.14],[9E9,9E9,9E9,9E9,9E9,9E9]],speeddata0,DefaultBlend,tool0;
  MoveAbsJ [[-3.02,33.53,23.96,10.61,5.23,-93.13],[9E9,9E9,9E9,9E9,9E9,9E9]],speeddata0,DefaultBlend,tool0;
  MoveAbsJ [[-2.71,33.59,23.86,10.45,5.67,-94.12],[9E9,9E9,9E9,9E9,9E9,9E9]],speeddata0,DefaultBlend,tool0;
  MoveAbsJ [[-2.40,33.64,23.76,10.30,6.11,-95.12],[9E9,9E9,9E9,9E9,9E9,9E9]],speeddata0,DefaultBlend,tool0;
  MoveAbsJ [[-2.09,33.69,23.66,10.14,6.55,-96.11],[9E9,9E9,9E9,9E9,9E9,9E9]],speeddata0,DefaultBlend,tool0;
  MoveAbsJ [[-1.78,33.74,23.57,9.99,7.00,-97.10],[9E9,9E9,9E9,9E9,9E9,9E9]],speeddata0,DefaultBlend,tool0;
  MoveAbsJ [[-1.47,33.80,23.47,9.84,7.44,-98.09],[9E9,9E9,9E9,9E9,9E9,9E9]],speeddata0,DefaultBlend,tool0;
  MoveAbsJ [[-1.16,33.85,23.37,9.68,7.88,-99.08],[9E9,9E9,9E9,9E9,9E9,9E9]],speeddata0,DefaultBlend,tool0;
  MoveAbsJ [[-0.85,33.90,23.27,9.53,8.32,-100.07],[9E9,9E9,9E9,9E9,9E9,9E9]],speeddata0,DefaultBlend,tool0;
  MoveAbsJ [[-0.53,33.95,23.17,9.38,8.76,-101.07],[9E9,9E9,9E9,9E9,9E9,9E9]],speeddata0,DefaultBlend,tool0;
  MoveAbsJ [[-0.22,34.01,23.08,9.22,9.20,-102.06],[9E9,9E9,9E9,9E9,9E9,9E9]],speeddata0,DefaultBlend,tool0;
  MoveAbsJ [[0.09,34.06,22.98,9.07,9.64,-103.05],[9E9,9E9,9E9,9E9,9E9,9E9]],speeddata0,DefaultBlend,tool0;
  MoveAbsJ [[0.40,34.11,22.88,8.91,10.08,-104.04],[9E9,9E9,9E9,9E9,9E9,9E9]],speeddata0,DefaultBlend,tool0;
  MoveAbsJ [[0.71,34.16,22.78,8.76,10.52,-105.03],[9E9,9E9,9E9,9E9,9E9,9E9]],speeddata0,DefaultBlend,tool0;
  MoveAbsJ [[1.02,34.22,22.68,8.61,10.96,-106.03],[9E9,9E9,9E9,9E9,9E9,9E9]],speeddata0,DefaultBlend,tool0;
  MoveAbsJ [[1.33,34.27,22.59,8.45,11.40,-107.02],[9E9,9E9,9E9,9E9,9E9,9E9]],speeddata0,DefaultBlend,tool0;
  MoveAbsJ [[1.64,34.32,22.49,8.30,11.84,-108.01],[9E9,9E9,9E9,9E9,9E9,9E9]],speeddata0,DefaultBlend,tool0;
  MoveAbsJ [[1.95,34.37,22.39,8.15,12.28,-109.00],[9E9,9E9,9E9,9E9,9E9,9E9]],speeddata0,DefaultBlend,tool0;
  MoveAbsJ [[2.26,34.43,22.29,7.99,12.72,-109.99],[9E9,9E9,9E9,9E9,9E9,9E9]],speeddata0,DefaultBlend,tool0;
  MoveAbsJ [[2.58,34.48,22.20,7.84,13.16,-110.98],[9E9,9E9,9E9,9E9,9E9,9E9]],speeddata0,DefaultBlend,tool0;
  MoveAbsJ [[2.89,34.53,22.10,7.69,13.61,-111.98],[9E9,9E9,9E9,9E9,9E9,9E9]],speeddata0,DefaultBlend,tool0;
  MoveAbsJ [[3.20,34.58,22.00,7.53,14.05,-112.97],[9E9,9E9,9E9,9E9,9E9,9E9]],speeddata0,DefaultBlend,tool0;
  MoveAbsJ [[3.51,34.64,21.90,7.38,14.49,-113.96],[9E9,9E9,9E9,9E9,9E9,9E9]],speeddata0,DefaultBlend,tool0;
  MoveAbsJ [[3.82,34.69,21.80,7.22,14.93,-114.95],[9E9,9E9,9E9,9E9,9E9,9E9]],speeddata0,DefaultBlend,tool0;
  MoveAbsJ [[4.13,34.74,21.71,7.07,15.37,-115.94],[9E9,9E9,9E9,9E9,9E9,9E9]],speeddata0,DefaultBlend,tool0;
  MoveAbsJ [[4.44,34.79,21.61,6.92,15.81,-116.94],[9E9,9E9,9E9,9E9,9E9,9E9]],speeddata0,DefaultBlend,tool0;
  MoveAbsJ [[4.75,34.85,21.51,6.76,16.25,-117.93],[9E9,9E9,9E9,9E9,9E9,9E9]],speeddata0,DefaultBlend,tool0;
  MoveAbsJ [[5.06,34.90,21.41,6.61,16.69,-118.92],[9E9,9E9,9E9,9E9,9E9,9E9]],speeddata0,DefaultBlend,tool0;
  MoveAbsJ [[5.37,34.95,21.31,6.46,17.13,-119.91],[9E9,9E9,9E9,9E9,9E9,9E9]],speeddata0,DefaultBlend,tool0;
  MoveAbsJ [[5.69,35.00,21.22,6.30,17.57,-120.90],[9E9,9E9,9E9,9E9,9E9,9E9]],speeddata0,DefaultBlend,tool0;
  MoveAbsJ [[6.00,35.06,21.12,6.15,18.01,-121.89],[9E9,9E9,9E9,9E9,9E9,9E9]],speeddata0,DefaultBlend,tool0;
  MoveAbsJ [[6.31,35.11,21.02,5.99,18.45,-122.89],[9E9,9E9,9E9,9E9,9E9,9E9]],speeddata0,DefaultBlend,tool0;
  MoveAbsJ [[6.62,35.16,20.92,5.84,18.89,-123.88],[9E9,9E9,9E9,9E9,9E9,9E9]],speeddata0,DefaultBlend,tool0;
  MoveAbsJ [[6.93,35.21,20.83,5.69,19.33,-124.87],[9E9,9E9,9E9,9E9,9E9,9E9]],speeddata0,DefaultBlend,tool0;
  MoveAbsJ [[7.24,35.27,20.73,5.53,19.77,-125.86],[9E9,9E9,9E9,9E9,9E9,9E9]],speeddata0,DefaultBlend,tool0;
  MoveAbsJ [[7.55,35.32,20.63,5.38,20.22,-126.85],[9E9,9E9,9E9,9E9,9E9,9E9]],speeddata0,DefaultBlend,tool0;
  MoveAbsJ [[7.86,35.37,20.53,5.23,20.66,-127.84],[9E9,9E9,9E9,9E9,9E9,9E9]],speeddata0,DefaultBlend,tool0;
  MoveAbsJ [[8.17,35.42,20.43,5.07,21.10,-128.84],[9E9,9E9,9E9,9E9,9E9,9E9]],speeddata0,DefaultBlend,tool0;
  MoveAbsJ [[8.48,35.48,20.34,4.92,21.54,-129.83],[9E9,9E9,9E9,9E9,9E9,9E9]],speeddata0,DefaultBlend,tool0;
  MoveAbsJ [[8.79,35.53,20.24,4.76,21.98,-130.82],[9E9,9E9,9E9,9E9,9E9,9E9]],speeddata0,DefaultBlend,tool0;
  MoveAbsJ [[9.11,35.58,20.14,4.61,22.42,-131.81],[9E9,9E9,9E9,9E9,9E9,9E9]],speeddata0,DefaultBlend,tool0;
  MoveAbsJ [[9.42,35.63,20.04,4.46,22.86,-132.80],[9E9,9E9,9E9,9E9,9E9,9E9]],speeddata0,DefaultBlend,tool0;
  MoveAbsJ [[9.73,35.69,19.95,4.30,23.30,-133.80],[9E9,9E9,9E9,9E9,9E9,9E9]],speeddata0,DefaultBlend,tool0;
  MoveAbsJ [[10.04,35.74,19.85,4.15,23.74,-134.79],[9E9,9E9,9E9,9E9,9E9,9E9]],speeddata0,DefaultBlend,tool0;
  MoveAbsJ [[10.35,35.79,19.75,4.00,24.18,-135.78],[9E9,9E9,9E9,9E9,9E9,9E9]],speeddata0,DefaultBlend,tool0;
  MoveAbsJ [[10.66,35.84,19.65,3.84,24.62,-136.77],[9E9,9E9,9E9,9E9,9E9,9E9]],speeddata0,DefaultBlend,tool0;
  MoveAbsJ [[10.97,35.90,19.55,3.69,25.06,-137.76],[9E9,9E9,9E9,9E9,9E9,9E9]],speeddata0,DefaultBlend,tool0;
  MoveAbsJ [[11.28,35.95,19.46,3.54,25.50,-138.75],[9E9,9E9,9E9,9E9,9E9,9E9]],speeddata0,DefaultBlend,tool0;
  MoveAbsJ [[11.59,36.00,19.36,3.38,25.94,-139.75],[9E9,9E9,9E9,9E9,9E9,9E9]],speeddata0,DefaultBlend,tool0;
  MoveAbsJ [[11.90,36.05,19.26,3.23,26.38,-140.74],[9E9,9E9,9E9,9E9,9E9,9E9]],speeddata0,DefaultBlend,tool0;
  MoveAbsJ [[12.22,36.11,19.16,3.07,26.83,-141.73],[9E9,9E9,9E9,9E9,9E9,9E9]],speeddata0,DefaultBlend,tool0;
  MoveAbsJ [[12.53,36.16,19.06,2.92,27.27,-142.72],[9E9,9E9,9E9,9E9,9E9,9E9]],speeddata0,DefaultBlend,tool0;
  MoveAbsJ [[12.84,36.21,18.97,2.77,27.71,-143.71],[9E9,9E9,9E9,9E9,9E9,9E9]],speeddata0,DefaultBlend,tool0;
  MoveAbsJ [[13.15,36.26,18.87,2.61,28.15,-144.70],[9E9,9E9,9E9,9E9,9E9,9E9]],speeddata0,DefaultBlend,tool0;
  MoveAbsJ [[13.46,36.32,18.77,2.46,28.59,-145.70],[9E9,9E9,9E9,9E9,9E9,9E9]],speeddata0,DefaultBlend,tool0;
  MoveAbsJ [[13.77,36.37,18.67,2.31,29.03,-146.69],[9E9,9E9,9E9,9E9,9E9,9E9]],speeddata0,DefaultBlend,tool0;
  MoveAbsJ [[14.08,36.42,18.58,2.15,29.47,-147.68],[9E9,9E9,9E9,9E9,9E9,9E9]],speeddata0,DefaultBlend,tool0;
  MoveAbsJ [[14.39,36.47,18.48,2.00,29.91,-148.67],[9E9,9E9,9E9,9E9,9E9,9E9]],speeddata0,DefaultBlend,tool0;
  MoveAbsJ [[14.70,36.53,18.38,1.84,30.35,-149.66],[9E9,9E9,9E9,9E9,9E9,9E9]],speeddata0,DefaultBlend,tool0;
  MoveAbsJ [[15.01,36.58,18.28,1.69,30.79,-150.66],[9E9,9E9,9E9,9E9,9E9,9E9]],speeddata0,DefaultBlend,tool0;
  MoveAbsJ [[15.33,36.63,18.18,1.54,31.23,-151.65],[9E9,9E9,9E9,9E9,9E9,9E9]],speeddata0,DefaultBlend,tool0;
  MoveAbsJ [[15.64,36.68,18.09,1.38,31.67,-152.64],[9E9,9E9,9E9,9E9,9E9,9E9]],speeddata0,DefaultBlend,tool0;
  MoveAbsJ [[15.95,36.74,17.99,1.23,32.11,-153.63],[9E9,9E9,9E9,9E9,9E9,9E9]],speeddata0,DefaultBlend,tool0;
  MoveAbsJ [[16.26,36.79,17.89,1.08,32.55,-154.62],[9E9,9E9,9E9,9E9,9E9,9E9]],speeddata0,DefaultBlend,tool0;
  MoveAbsJ [[16.57,36.84,17.79,0.92,32.99,-155.61],[9E9,9E9,9E9,9E9,9E9,9E9]],speeddata0,DefaultBlend,tool0;
  MoveAbsJ [[16.88,36.89,17.69,0.77,33.43,-156.61],[9E9,9E9,9E9,9E9,9E9,9E9]],speeddata0,DefaultBlend,tool0;
  MoveAbsJ [[17.19,36.95,17.60,0.61,33.88,-157.60],[9E9,9E9,9E9,9E9,9E9,9E9]],speeddata0,DefaultBlend,tool0;
  MoveAbsJ [[17.50,37.00,17.50,0.46,34.32,-158.59],[9E9,9E9,9E9,9E9,9E9,9E9]],speeddata0,DefaultBlend,tool0;
  MoveAbsJ [[17.81,37.05,17.40,0.31,34.76,-159.58],[9E9,9E9,9E9,9E9,9E9,9E9]],speeddata0,DefaultBlend,tool0;
  MoveAbsJ [[18.12,37.10,17.30,0.15,35.20,-160.57],[9E9,9E9,9E9,9E9,9E9,9E9]],speeddata0,DefaultBlend,tool0;
  MoveAbsJ [[18.43,37.16,17.21,-0.00,35.64,-161.56],[9E9,9E9,9E9,9E9,9E9,9E9]],speeddata0,FinePoint,tool0;
  TPWrite "Action 4 LinearMovement.";
  MoveAbsJ [[18.43,37.16,17.21,-0.00,35.64,-161.56],[9E9,9E9,9E9,9E9,9E9,9E9]],speeddata0,DefaultBlend,tool0;
  MoveAbsJ [[18.43,37.97,17.26,-0.00,34.77,-161.57],[9E9,9E9,9E9,9E9,9E9,9E9]],speeddata0,DefaultBlend,tool0;
  MoveAbsJ [[18.43,38.79,17.32,-0.00,33.90,-161.57],[9E9,9E9,9E9,9E9,9E9,9E9]],speeddata0,DefaultBlend,tool0;
  MoveAbsJ [[18.43,39.62,17.35,-0.00,33.03,-161.57],[9E9,9E9,9E9,9E9,9E9,9E9]],speeddata0,DefaultBlend,tool0;
  MoveAbsJ [[18.43,40.46,17.36,-0.00,32.18,-161.57],[9E9,9E9,9E9,9E9,9E9,9E9]],speeddata0,DefaultBlend,tool0;
  MoveAbsJ [[18.43,41.32,17.35,-0.00,31.33,-161.57],[9E9,9E9,9E9,9E9,9E9,9E9]],speeddata0,DefaultBlend,tool0;
  MoveAbsJ [[18.43,42.19,17.31,-0.00,30.50,-161.57],[9E9,9E9,9E9,9E9,9E9,9E9]],speeddata0,DefaultBlend,tool0;
  MoveAbsJ [[18.43,43.07,17.25,-0.00,29.67,-161.57],[9E9,9E9,9E9,9E9,9E9,9E9]],speeddata0,DefaultBlend,tool0;
  MoveAbsJ [[18.43,43.97,17.17,-0.00,28.86,-161.57],[9E9,9E9,9E9,9E9,9E9,9E9]],speeddata0,FinePoint,tool0;
  TPWrite "Action 5 OpenGripper.";
  TPWrite "Press Play to Continue";
  Stop;
  TPWrite "Action 6 LinearMovement.";
  MoveAbsJ [[18.43,43.97,17.17,-0.00,28.86,-161.57],[9E9,9E9,9E9,9E9,9E9,9E9]],speeddata0,DefaultBlend,tool0;
  MoveAbsJ [[18.43,43.09,17.24,-0.00,29.67,-161.57],[9E9,9E9,9E9,9E9,9E9,9E9]],speeddata0,DefaultBlend,tool0;
  MoveAbsJ [[18.43,42.21,17.30,-0.00,30.49,-161.57],[9E9,9E9,9E9,9E9,9E9,9E9]],speeddata0,DefaultBlend,tool0;
  MoveAbsJ [[18.43,41.33,17.34,-0.00,31.32,-161.57],[9E9,9E9,9E9,9E9,9E9,9E9]],speeddata0,DefaultBlend,tool0;
  MoveAbsJ [[18.43,40.48,17.36,0.00,32.16,-161.57],[9E9,9E9,9E9,9E9,9E9,9E9]],speeddata0,DefaultBlend,tool0;
  MoveAbsJ [[18.43,39.63,17.36,0.00,33.01,-161.57],[9E9,9E9,9E9,9E9,9E9,9E9]],speeddata0,DefaultBlend,tool0;
  MoveAbsJ [[18.43,38.79,17.33,0.00,33.88,-161.57],[9E9,9E9,9E9,9E9,9E9,9E9]],speeddata0,DefaultBlend,tool0;
  MoveAbsJ [[18.43,37.97,17.27,0.00,34.75,-161.57],[9E9,9E9,9E9,9E9,9E9,9E9]],speeddata0,DefaultBlend,tool0;
  MoveAbsJ [[18.43,37.16,17.20,0.00,35.64,-161.57],[9E9,9E9,9E9,9E9,9E9,9E9]],speeddata0,FinePoint,tool0;
  TPWrite "Action 7 FreeMovement.";
  MoveAbsJ [[18.43,37.16,17.20,0.00,35.64,-161.57],[9E9,9E9,9E9,9E9,9E9,9E9]],speeddata0,DefaultBlend,tool0;
  MoveAbsJ [[17.88,36.95,17.36,-0.99,35.76,-161.24],[9E9,9E9,9E9,9E9,9E9,9E9]],speeddata0,DefaultBlend,tool0;
  MoveAbsJ [[17.33,36.74,17.51,-1.98,35.88,-160.91],[9E9,9E9,9E9,9E9,9E9,9E9]],speeddata0,DefaultBlend,tool0;
  MoveAbsJ [[16.78,36.54,17.67,-2.96,36.00,-160.58],[9E9,9E9,9E9,9E9,9E9,9E9]],speeddata0,DefaultBlend,tool0;
  MoveAbsJ [[16.23,36.33,17.83,-3.95,36.12,-160.26],[9E9,9E9,9E9,9E9,9E9,9E9]],speeddata0,DefaultBlend,tool0;
  MoveAbsJ [[15.68,36.12,17.99,-4.94,36.24,-159.93],[9E9,9E9,9E9,9E9,9E9,9E9]],speeddata0,DefaultBlend,tool0;
  MoveAbsJ [[15.13,35.91,18.14,-5.93,36.36,-159.60],[9E9,9E9,9E9,9E9,9E9,9E9]],speeddata0,DefaultBlend,tool0;
  MoveAbsJ [[14.58,35.70,18.30,-6.91,36.48,-159.28],[9E9,9E9,9E9,9E9,9E9,9E9]],speeddata0,DefaultBlend,tool0;
  MoveAbsJ [[14.03,35.49,18.46,-7.90,36.60,-158.95],[9E9,9E9,9E9,9E9,9E9,9E9]],speeddata0,DefaultBlend,tool0;
  MoveAbsJ [[13.48,35.28,18.62,-8.89,36.72,-158.62],[9E9,9E9,9E9,9E9,9E9,9E9]],speeddata0,DefaultBlend,tool0;
  MoveAbsJ [[12.93,35.07,18.77,-9.88,36.84,-158.30],[9E9,9E9,9E9,9E9,9E9,9E9]],speeddata0,DefaultBlend,tool0;
  MoveAbsJ [[12.38,34.86,18.93,-10.87,36.96,-157.97],[9E9,9E9,9E9,9E9,9E9,9E9]],speeddata0,DefaultBlend,tool0;
  MoveAbsJ [[11.83,34.65,19.09,-11.85,37.08,-157.64],[9E9,9E9,9E9,9E9,9E9,9E9]],speeddata0,DefaultBlend,tool0;
  MoveAbsJ [[11.28,34.44,19.25,-12.84,37.20,-157.32],[9E9,9E9,9E9,9E9,9E9,9E9]],speeddata0,DefaultBlend,tool0;
  MoveAbsJ [[10.73,34.23,19.40,-13.83,37.32,-156.99],[9E9,9E9,9E9,9E9,9E9,9E9]],speeddata0,DefaultBlend,tool0;
  MoveAbsJ [[10.17,34.02,19.56,-14.82,37.44,-156.66],[9E9,9E9,9E9,9E9,9E9,9E9]],speeddata0,DefaultBlend,tool0;
  MoveAbsJ [[9.62,33.81,19.72,-15.80,37.56,-156.34],[9E9,9E9,9E9,9E9,9E9,9E9]],speeddata0,DefaultBlend,tool0;
  MoveAbsJ [[9.07,33.60,19.88,-16.79,37.68,-156.01],[9E9,9E9,9E9,9E9,9E9,9E9]],speeddata0,DefaultBlend,tool0;
  MoveAbsJ [[8.52,33.39,20.03,-17.78,37.80,-155.68],[9E9,9E9,9E9,9E9,9E9,9E9]],speeddata0,DefaultBlend,tool0;
  MoveAbsJ [[7.97,33.18,20.19,-18.77,37.92,-155.36],[9E9,9E9,9E9,9E9,9E9,9E9]],speeddata0,DefaultBlend,tool0;
  MoveAbsJ [[7.42,32.97,20.35,-19.75,38.04,-155.03],[9E9,9E9,9E9,9E9,9E9,9E9]],speeddata0,DefaultBlend,tool0;
  MoveAbsJ [[6.87,32.76,20.51,-20.74,38.16,-154.70],[9E9,9E9,9E9,9E9,9E9,9E9]],speeddata0,DefaultBlend,tool0;
  MoveAbsJ [[6.32,32.55,20.66,-21.73,38.28,-154.38],[9E9,9E9,9E9,9E9,9E9,9E9]],speeddata0,DefaultBlend,tool0;
  MoveAbsJ [[5.77,32.34,20.82,-22.72,38.40,-154.05],[9E9,9E9,9E9,9E9,9E9,9E9]],speeddata0,DefaultBlend,tool0;
  MoveAbsJ [[5.22,32.13,20.98,-23.71,38.52,-153.72],[9E9,9E9,9E9,9E9,9E9,9E9]],speeddata0,DefaultBlend,tool0;
  MoveAbsJ [[4.67,31.93,21.14,-24.69,38.64,-153.40],[9E9,9E9,9E9,9E9,9E9,9E9]],speeddata0,DefaultBlend,tool0;
  MoveAbsJ [[4.12,31.72,21.29,-25.68,38.76,-153.07],[9E9,9E9,9E9,9E9,9E9,9E9]],speeddata0,DefaultBlend,tool0;
  MoveAbsJ [[3.57,31.51,21.45,-26.67,38.88,-152.74],[9E9,9E9,9E9,9E9,9E9,9E9]],speeddata0,DefaultBlend,tool0;
  MoveAbsJ [[3.02,31.30,21.61,-27.66,39.00,-152.42],[9E9,9E9,9E9,9E9,9E9,9E9]],speeddata0,DefaultBlend,tool0;
  MoveAbsJ [[2.47,31.09,21.77,-28.64,39.12,-152.09],[9E9,9E9,9E9,9E9,9E9,9E9]],speeddata0,DefaultBlend,tool0;
  MoveAbsJ [[1.91,30.88,21.92,-29.63,39.24,-151.76],[9E9,9E9,9E9,9E9,9E9,9E9]],speeddata0,DefaultBlend,tool0;
  MoveAbsJ [[1.36,30.67,22.08,-30.62,39.36,-151.44],[9E9,9E9,9E9,9E9,9E9,9E9]],speeddata0,DefaultBlend,tool0;
  MoveAbsJ [[0.81,30.46,22.24,-31.61,39.48,-151.11],[9E9,9E9,9E9,9E9,9E9,9E9]],speeddata0,DefaultBlend,tool0;
  MoveAbsJ [[0.26,30.25,22.40,-32.60,39.60,-150.78],[9E9,9E9,9E9,9E9,9E9,9E9]],speeddata0,DefaultBlend,tool0;
  MoveAbsJ [[-0.29,30.04,22.55,-33.58,39.72,-150.46],[9E9,9E9,9E9,9E9,9E9,9E9]],speeddata0,DefaultBlend,tool0;
  MoveAbsJ [[-0.84,29.83,22.71,-34.57,39.84,-150.13],[9E9,9E9,9E9,9E9,9E9,9E9]],speeddata0,DefaultBlend,tool0;
  MoveAbsJ [[-1.39,29.62,22.87,-35.56,39.96,-149.80],[9E9,9E9,9E9,9E9,9E9,9E9]],speeddata0,DefaultBlend,tool0;
  MoveAbsJ [[-1.94,29.41,23.02,-36.55,40.08,-149.48],[9E9,9E9,9E9,9E9,9E9,9E9]],speeddata0,DefaultBlend,tool0;
  MoveAbsJ [[-2.49,29.20,23.18,-37.53,40.20,-149.15],[9E9,9E9,9E9,9E9,9E9,9E9]],speeddata0,DefaultBlend,tool0;
  MoveAbsJ [[-3.04,28.99,23.34,-38.52,40.32,-148.82],[9E9,9E9,9E9,9E9,9E9,9E9]],speeddata0,DefaultBlend,tool0;
  MoveAbsJ [[-3.59,28.78,23.50,-39.51,40.44,-148.50],[9E9,9E9,9E9,9E9,9E9,9E9]],speeddata0,DefaultBlend,tool0;
  MoveAbsJ [[-4.14,28.57,23.65,-40.50,40.56,-148.17],[9E9,9E9,9E9,9E9,9E9,9E9]],speeddata0,DefaultBlend,tool0;
  MoveAbsJ [[-4.69,28.36,23.81,-41.48,40.68,-147.84],[9E9,9E9,9E9,9E9,9E9,9E9]],speeddata0,DefaultBlend,tool0;
  MoveAbsJ [[-5.24,28.15,23.97,-42.47,40.80,-147.52],[9E9,9E9,9E9,9E9,9E9,9E9]],speeddata0,DefaultBlend,tool0;
  MoveAbsJ [[-5.80,27.94,24.13,-43.46,40.92,-147.19],[9E9,9E9,9E9,9E9,9E9,9E9]],speeddata0,DefaultBlend,tool0;
  MoveAbsJ [[-6.35,27.73,24.28,-44.45,41.04,-146.86],[9E9,9E9,9E9,9E9,9E9,9E9]],speeddata0,DefaultBlend,tool0;
  MoveAbsJ [[-6.90,27.52,24.44,-45.44,41.16,-146.54],[9E9,9E9,9E9,9E9,9E9,9E9]],speeddata0,DefaultBlend,tool0;
  MoveAbsJ [[-7.45,27.31,24.60,-46.42,41.28,-146.21],[9E9,9E9,9E9,9E9,9E9,9E9]],speeddata0,DefaultBlend,tool0;
  MoveAbsJ [[-8.00,27.11,24.76,-47.41,41.40,-145.88],[9E9,9E9,9E9,9E9,9E9,9E9]],speeddata0,DefaultBlend,tool0;
  MoveAbsJ [[-8.55,26.90,24.91,-48.40,41.52,-145.56],[9E9,9E9,9E9,9E9,9E9,9E9]],speeddata0,DefaultBlend,tool0;
  MoveAbsJ [[-9.10,26.69,25.07,-49.39,41.64,-145.23],[9E9,9E9,9E9,9E9,9E9,9E9]],speeddata0,DefaultBlend,tool0;
  MoveAbsJ [[-9.65,26.48,25.23,-50.37,41.76,-144.90],[9E9,9E9,9E9,9E9,9E9,9E9]],speeddata0,DefaultBlend,tool0;
  MoveAbsJ [[-10.20,26.27,25.39,-51.36,41.88,-144.58],[9E9,9E9,9E9,9E9,9E9,9E9]],speeddata0,DefaultBlend,tool0;
  MoveAbsJ [[-10.75,26.06,25.54,-52.35,42.00,-144.25],[9E9,9E9,9E9,9E9,9E9,9E9]],speeddata0,DefaultBlend,tool0;
  MoveAbsJ [[-11.30,25.85,25.70,-53.34,42.12,-143.92],[9E9,9E9,9E9,9E9,9E9,9E9]],speeddata0,DefaultBlend,tool0;
  MoveAbsJ [[-11.85,25.64,25.86,-54.33,42.24,-143.60],[9E9,9E9,9E9,9E9,9E9,9E9]],speeddata0,DefaultBlend,tool0;
  MoveAbsJ [[-12.40,25.43,26.02,-55.31,42.36,-143.27],[9E9,9E9,9E9,9E9,9E9,9E9]],speeddata0,DefaultBlend,tool0;
  MoveAbsJ [[-12.95,25.22,26.17,-56.30,42.49,-142.94],[9E9,9E9,9E9,9E9,9E9,9E9]],speeddata0,DefaultBlend,tool0;
  MoveAbsJ [[-13.50,25.01,26.33,-57.29,42.61,-142.62],[9E9,9E9,9E9,9E9,9E9,9E9]],speeddata0,DefaultBlend,tool0;
  MoveAbsJ [[-14.06,24.80,26.49,-58.28,42.73,-142.29],[9E9,9E9,9E9,9E9,9E9,9E9]],speeddata0,DefaultBlend,tool0;
  MoveAbsJ [[-14.61,24.59,26.65,-59.26,42.85,-141.96],[9E9,9E9,9E9,9E9,9E9,9E9]],speeddata0,DefaultBlend,tool0;
  MoveAbsJ [[-15.16,24.38,26.80,-60.25,42.97,-141.64],[9E9,9E9,9E9,9E9,9E9,9E9]],speeddata0,DefaultBlend,tool0;
  MoveAbsJ [[-15.71,24.17,26.96,-61.24,43.09,-141.31],[9E9,9E9,9E9,9E9,9E9,9E9]],speeddata0,DefaultBlend,tool0;
  MoveAbsJ [[-16.26,23.96,27.12,-62.23,43.21,-140.98],[9E9,9E9,9E9,9E9,9E9,9E9]],speeddata0,DefaultBlend,tool0;
  MoveAbsJ [[-16.81,23.75,27.28,-63.22,43.33,-140.66],[9E9,9E9,9E9,9E9,9E9,9E9]],speeddata0,DefaultBlend,tool0;
  MoveAbsJ [[-17.36,23.54,27.43,-64.20,43.45,-140.33],[9E9,9E9,9E9,9E9,9E9,9E9]],speeddata0,DefaultBlend,tool0;
  MoveAbsJ [[-17.91,23.33,27.59,-65.19,43.57,-140.00],[9E9,9E9,9E9,9E9,9E9,9E9]],speeddata0,DefaultBlend,tool0;
  MoveAbsJ [[-18.46,23.12,27.75,-66.18,43.69,-139.68],[9E9,9E9,9E9,9E9,9E9,9E9]],speeddata0,DefaultBlend,tool0;
  MoveAbsJ [[-19.01,22.91,27.91,-67.17,43.81,-139.35],[9E9,9E9,9E9,9E9,9E9,9E9]],speeddata0,DefaultBlend,tool0;
  MoveAbsJ [[-19.56,22.70,28.06,-68.15,43.93,-139.02],[9E9,9E9,9E9,9E9,9E9,9E9]],speeddata0,DefaultBlend,tool0;
  MoveAbsJ [[-20.11,22.50,28.22,-69.14,44.05,-138.70],[9E9,9E9,9E9,9E9,9E9,9E9]],speeddata0,DefaultBlend,tool0;
  MoveAbsJ [[-20.66,22.29,28.38,-70.13,44.17,-138.37],[9E9,9E9,9E9,9E9,9E9,9E9]],speeddata0,DefaultBlend,tool0;
  MoveAbsJ [[-21.21,22.08,28.54,-71.12,44.29,-138.04],[9E9,9E9,9E9,9E9,9E9,9E9]],speeddata0,DefaultBlend,tool0;
  MoveAbsJ [[-21.77,21.87,28.69,-72.10,44.41,-137.72],[9E9,9E9,9E9,9E9,9E9,9E9]],speeddata0,DefaultBlend,tool0;
  MoveAbsJ [[-22.32,21.66,28.85,-73.09,44.53,-137.39],[9E9,9E9,9E9,9E9,9E9,9E9]],speeddata0,DefaultBlend,tool0;
  MoveAbsJ [[-22.87,21.45,29.01,-74.08,44.65,-137.06],[9E9,9E9,9E9,9E9,9E9,9E9]],speeddata0,DefaultBlend,tool0;
  MoveAbsJ [[-23.42,21.24,29.17,-75.07,44.77,-136.74],[9E9,9E9,9E9,9E9,9E9,9E9]],speeddata0,DefaultBlend,tool0;
  MoveAbsJ [[-23.97,21.03,29.32,-76.06,44.89,-136.41],[9E9,9E9,9E9,9E9,9E9,9E9]],speeddata0,DefaultBlend,tool0;
  MoveAbsJ [[-24.52,20.82,29.48,-77.04,45.01,-136.08],[9E9,9E9,9E9,9E9,9E9,9E9]],speeddata0,DefaultBlend,tool0;
  MoveAbsJ [[-25.07,20.61,29.64,-78.03,45.13,-135.75],[9E9,9E9,9E9,9E9,9E9,9E9]],speeddata0,DefaultBlend,tool0;
  MoveAbsJ [[-25.62,20.40,29.80,-79.02,45.25,-135.43],[9E9,9E9,9E9,9E9,9E9,9E9]],speeddata0,DefaultBlend,tool0;
  MoveAbsJ [[-26.17,20.19,29.95,-80.01,45.37,-135.10],[9E9,9E9,9E9,9E9,9E9,9E9]],speeddata0,DefaultBlend,tool0;
  MoveAbsJ [[-26.72,19.98,30.11,-80.99,45.49,-134.77],[9E9,9E9,9E9,9E9,9E9,9E9]],speeddata0,DefaultBlend,tool0;
  MoveAbsJ [[-27.27,19.77,30.27,-81.98,45.61,-134.45],[9E9,9E9,9E9,9E9,9E9,9E9]],speeddata0,DefaultBlend,tool0;
  MoveAbsJ [[-27.82,19.56,30.43,-82.97,45.73,-134.12],[9E9,9E9,9E9,9E9,9E9,9E9]],speeddata0,DefaultBlend,tool0;
  MoveAbsJ [[-28.37,19.35,30.58,-83.96,45.85,-133.79],[9E9,9E9,9E9,9E9,9E9,9E9]],speeddata0,DefaultBlend,tool0;
  MoveAbsJ [[-28.92,19.14,30.74,-84.95,45.97,-133.47],[9E9,9E9,9E9,9E9,9E9,9E9]],speeddata0,DefaultBlend,tool0;
  MoveAbsJ [[-29.47,18.93,30.90,-85.93,46.09,-133.14],[9E9,9E9,9E9,9E9,9E9,9E9]],speeddata0,DefaultBlend,tool0;
  MoveAbsJ [[-30.03,18.72,31.06,-86.92,46.21,-132.81],[9E9,9E9,9E9,9E9,9E9,9E9]],speeddata0,DefaultBlend,tool0;
  MoveAbsJ [[-30.58,18.51,31.21,-87.91,46.33,-132.49],[9E9,9E9,9E9,9E9,9E9,9E9]],speeddata0,DefaultBlend,tool0;
  MoveAbsJ [[-31.13,18.30,31.37,-88.90,46.45,-132.16],[9E9,9E9,9E9,9E9,9E9,9E9]],speeddata0,DefaultBlend,tool0;
  MoveAbsJ [[-31.68,18.09,31.53,-89.88,46.57,-131.83],[9E9,9E9,9E9,9E9,9E9,9E9]],speeddata0,DefaultBlend,tool0;
  MoveAbsJ [[-32.23,17.88,31.69,-90.87,46.69,-131.51],[9E9,9E9,9E9,9E9,9E9,9E9]],speeddata0,DefaultBlend,tool0;
  MoveAbsJ [[-32.78,17.68,31.84,-91.86,46.81,-131.18],[9E9,9E9,9E9,9E9,9E9,9E9]],speeddata0,DefaultBlend,tool0;
  MoveAbsJ [[-33.33,17.47,32.00,-92.85,46.93,-130.85],[9E9,9E9,9E9,9E9,9E9,9E9]],speeddata0,DefaultBlend,tool0;
  MoveAbsJ [[-33.88,17.26,32.16,-93.84,47.05,-130.53],[9E9,9E9,9E9,9E9,9E9,9E9]],speeddata0,DefaultBlend,tool0;
  MoveAbsJ [[-34.43,17.05,32.32,-94.82,47.17,-130.20],[9E9,9E9,9E9,9E9,9E9,9E9]],speeddata0,DefaultBlend,tool0;
  MoveAbsJ [[-34.98,16.84,32.47,-95.81,47.29,-129.87],[9E9,9E9,9E9,9E9,9E9,9E9]],speeddata0,DefaultBlend,tool0;
  MoveAbsJ [[-35.53,16.63,32.63,-96.80,47.41,-129.55],[9E9,9E9,9E9,9E9,9E9,9E9]],speeddata0,DefaultBlend,tool0;
  MoveAbsJ [[-36.08,16.42,32.79,-97.79,47.53,-129.22],[9E9,9E9,9E9,9E9,9E9,9E9]],speeddata0,DefaultBlend,tool0;
  MoveAbsJ [[-36.63,16.21,32.95,-98.77,47.65,-128.89],[9E9,9E9,9E9,9E9,9E9,9E9]],speeddata0,DefaultBlend,tool0;
  MoveAbsJ [[-37.18,16.00,33.10,-99.76,47.77,-128.57],[9E9,9E9,9E9,9E9,9E9,9E9]],speeddata0,DefaultBlend,tool0;
  MoveAbsJ [[-37.73,15.79,33.26,-100.75,47.89,-128.24],[9E9,9E9,9E9,9E9,9E9,9E9]],speeddata0,DefaultBlend,tool0;
  MoveAbsJ [[-38.29,15.58,33.42,-101.74,48.01,-127.91],[9E9,9E9,9E9,9E9,9E9,9E9]],speeddata0,DefaultBlend,tool0;
  MoveAbsJ [[-38.84,15.37,33.58,-102.72,48.13,-127.59],[9E9,9E9,9E9,9E9,9E9,9E9]],speeddata0,DefaultBlend,tool0;
  MoveAbsJ [[-39.39,15.16,33.73,-103.71,48.25,-127.26],[9E9,9E9,9E9,9E9,9E9,9E9]],speeddata0,DefaultBlend,tool0;
  MoveAbsJ [[-39.94,14.95,33.89,-104.70,48.37,-126.93],[9E9,9E9,9E9,9E9,9E9,9E9]],speeddata0,DefaultBlend,tool0;
  MoveAbsJ [[-40.49,14.74,34.05,-105.69,48.49,-126.61],[9E9,9E9,9E9,9E9,9E9,9E9]],speeddata0,DefaultBlend,tool0;
  MoveAbsJ [[-41.04,14.53,34.21,-106.68,48.61,-126.28],[9E9,9E9,9E9,9E9,9E9,9E9]],speeddata0,DefaultBlend,tool0;
  MoveAbsJ [[-41.59,14.32,34.36,-107.66,48.73,-125.95],[9E9,9E9,9E9,9E9,9E9,9E9]],speeddata0,DefaultBlend,tool0;
  MoveAbsJ [[-42.14,14.11,34.52,-108.65,48.85,-125.63],[9E9,9E9,9E9,9E9,9E9,9E9]],speeddata0,DefaultBlend,tool0;
  MoveAbsJ [[-42.69,13.90,34.68,-109.64,48.97,-125.30],[9E9,9E9,9E9,9E9,9E9,9E9]],speeddata0,DefaultBlend,tool0;
  MoveAbsJ [[-43.24,13.69,34.84,-110.63,49.09,-124.97],[9E9,9E9,9E9,9E9,9E9,9E9]],speeddata0,DefaultBlend,tool0;
  MoveAbsJ [[-43.79,13.48,34.99,-111.61,49.21,-124.65],[9E9,9E9,9E9,9E9,9E9,9E9]],speeddata0,DefaultBlend,tool0;
  MoveAbsJ [[-44.34,13.27,35.15,-112.60,49.33,-124.32],[9E9,9E9,9E9,9E9,9E9,9E9]],speeddata0,DefaultBlend,tool0;
  MoveAbsJ [[-44.89,13.07,35.31,-113.59,49.45,-123.99],[9E9,9E9,9E9,9E9,9E9,9E9]],speeddata0,DefaultBlend,tool0;
  MoveAbsJ [[-45.44,12.86,35.47,-114.58,49.57,-123.67],[9E9,9E9,9E9,9E9,9E9,9E9]],speeddata0,DefaultBlend,tool0;
  MoveAbsJ [[-46.00,12.65,35.62,-115.57,49.70,-123.34],[9E9,9E9,9E9,9E9,9E9,9E9]],speeddata0,DefaultBlend,tool0;
  MoveAbsJ [[-46.55,12.44,35.78,-116.55,49.82,-123.01],[9E9,9E9,9E9,9E9,9E9,9E9]],speeddata0,DefaultBlend,tool0;
  MoveAbsJ [[-47.10,12.23,35.94,-117.54,49.94,-122.69],[9E9,9E9,9E9,9E9,9E9,9E9]],speeddata0,DefaultBlend,tool0;
  MoveAbsJ [[-47.65,12.02,36.09,-118.53,50.06,-122.36],[9E9,9E9,9E9,9E9,9E9,9E9]],speeddata0,DefaultBlend,tool0;
  MoveAbsJ [[-48.20,11.81,36.25,-119.52,50.18,-122.03],[9E9,9E9,9E9,9E9,9E9,9E9]],speeddata0,DefaultBlend,tool0;
  MoveAbsJ [[-48.75,11.60,36.41,-120.50,50.30,-121.71],[9E9,9E9,9E9,9E9,9E9,9E9]],speeddata0,DefaultBlend,tool0;
  MoveAbsJ [[-49.30,11.39,36.57,-121.49,50.42,-121.38],[9E9,9E9,9E9,9E9,9E9,9E9]],speeddata0,DefaultBlend,tool0;
  MoveAbsJ [[-49.85,11.18,36.72,-122.48,50.54,-121.05],[9E9,9E9,9E9,9E9,9E9,9E9]],speeddata0,DefaultBlend,tool0;
  MoveAbsJ [[-50.40,10.97,36.88,-123.47,50.66,-120.73],[9E9,9E9,9E9,9E9,9E9,9E9]],speeddata0,DefaultBlend,tool0;
  MoveAbsJ [[-50.95,10.76,37.04,-124.45,50.78,-120.40],[9E9,9E9,9E9,9E9,9E9,9E9]],speeddata0,DefaultBlend,tool0;
  MoveAbsJ [[-51.50,10.55,37.20,-125.44,50.90,-120.07],[9E9,9E9,9E9,9E9,9E9,9E9]],speeddata0,DefaultBlend,tool0;
  MoveAbsJ [[-52.05,10.34,37.35,-126.43,51.02,-119.75],[9E9,9E9,9E9,9E9,9E9,9E9]],speeddata0,DefaultBlend,tool0;
  MoveAbsJ [[-52.60,10.13,37.51,-127.42,51.14,-119.42],[9E9,9E9,9E9,9E9,9E9,9E9]],speeddata0,DefaultBlend,tool0;
  MoveAbsJ [[-53.15,9.92,37.67,-128.41,51.26,-119.09],[9E9,9E9,9E9,9E9,9E9,9E9]],speeddata0,DefaultBlend,tool0;
  MoveAbsJ [[-53.70,9.71,37.83,-129.39,51.38,-118.77],[9E9,9E9,9E9,9E9,9E9,9E9]],speeddata0,DefaultBlend,tool0;
  MoveAbsJ [[-54.26,9.50,37.98,-130.38,51.50,-118.44],[9E9,9E9,9E9,9E9,9E9,9E9]],speeddata0,DefaultBlend,tool0;
  MoveAbsJ [[-54.81,9.29,38.14,-131.37,51.62,-118.11],[9E9,9E9,9E9,9E9,9E9,9E9]],speeddata0,DefaultBlend,tool0;
  MoveAbsJ [[-55.36,9.08,38.30,-132.36,51.74,-117.79],[9E9,9E9,9E9,9E9,9E9,9E9]],speeddata0,DefaultBlend,tool0;
  MoveAbsJ [[-55.91,8.87,38.46,-133.34,51.86,-117.46],[9E9,9E9,9E9,9E9,9E9,9E9]],speeddata0,DefaultBlend,tool0;
  MoveAbsJ [[-56.46,8.66,38.61,-134.33,51.98,-117.13],[9E9,9E9,9E9,9E9,9E9,9E9]],speeddata0,DefaultBlend,tool0;
  MoveAbsJ [[-57.01,8.45,38.77,-135.32,52.10,-116.81],[9E9,9E9,9E9,9E9,9E9,9E9]],speeddata0,DefaultBlend,tool0;
  MoveAbsJ [[-57.56,8.25,38.93,-136.31,52.22,-116.48],[9E9,9E9,9E9,9E9,9E9,9E9]],speeddata0,DefaultBlend,tool0;
  MoveAbsJ [[-58.11,8.04,39.09,-137.30,52.34,-116.15],[9E9,9E9,9E9,9E9,9E9,9E9]],speeddata0,DefaultBlend,tool0;
  MoveAbsJ [[-58.66,7.83,39.24,-138.28,52.46,-115.83],[9E9,9E9,9E9,9E9,9E9,9E9]],speeddata0,DefaultBlend,tool0;
  MoveAbsJ [[-59.21,7.62,39.40,-139.27,52.58,-115.50],[9E9,9E9,9E9,9E9,9E9,9E9]],speeddata0,DefaultBlend,tool0;
  MoveAbsJ [[-59.76,7.41,39.56,-140.26,52.70,-115.17],[9E9,9E9,9E9,9E9,9E9,9E9]],speeddata0,DefaultBlend,tool0;
  MoveAbsJ [[-60.31,7.20,39.72,-141.25,52.82,-114.85],[9E9,9E9,9E9,9E9,9E9,9E9]],speeddata0,DefaultBlend,tool0;
  MoveAbsJ [[-60.86,6.99,39.87,-142.23,52.94,-114.52],[9E9,9E9,9E9,9E9,9E9,9E9]],speeddata0,DefaultBlend,tool0;
  MoveAbsJ [[-61.41,6.78,40.03,-143.22,53.06,-114.19],[9E9,9E9,9E9,9E9,9E9,9E9]],speeddata0,FinePoint,tool0;
  TPWrite "Action 8 LoadWorkpiece.";
  TPWrite "Press Play to Continue";
  Stop;
  TPWrite "Action 9 CloseGripper.";
  TPWrite "Press Play to Continue";
  Stop;
  TPWrite "Action 10 FreeMovement.";
  MoveAbsJ [[-61.41,6.78,40.03,-143.22,53.06,-114.19],[9E9,9E9,9E9,9E9,9E9,9E9]],speeddata0,DefaultBlend,tool0;
  MoveAbsJ [[-60.42,6.50,39.23,-142.58,52.48,-113.76],[9E9,9E9,9E9,9E9,9E9,9E9]],speeddata0,DefaultBlend,tool0;
  MoveAbsJ [[-59.42,6.23,38.43,-141.94,51.91,-113.34],[9E9,9E9,9E9,9E9,9E9,9E9]],speeddata0,DefaultBlend,tool0;
  MoveAbsJ [[-58.43,5.96,37.63,-141.30,51.33,-112.91],[9E9,9E9,9E9,9E9,9E9,9E9]],speeddata0,DefaultBlend,tool0;
  MoveAbsJ [[-57.43,5.68,36.83,-140.66,50.76,-112.48],[9E9,9E9,9E9,9E9,9E9,9E9]],speeddata0,DefaultBlend,tool0;
  MoveAbsJ [[-56.44,5.41,36.03,-140.03,50.18,-112.05],[9E9,9E9,9E9,9E9,9E9,9E9]],speeddata0,DefaultBlend,tool0;
  MoveAbsJ [[-55.44,5.13,35.23,-139.39,49.60,-111.63],[9E9,9E9,9E9,9E9,9E9,9E9]],speeddata0,DefaultBlend,tool0;
  MoveAbsJ [[-54.45,4.86,34.42,-138.75,49.03,-111.20],[9E9,9E9,9E9,9E9,9E9,9E9]],speeddata0,DefaultBlend,tool0;
  MoveAbsJ [[-53.45,4.58,33.62,-138.11,48.45,-110.77],[9E9,9E9,9E9,9E9,9E9,9E9]],speeddata0,DefaultBlend,tool0;
  MoveAbsJ [[-52.46,4.31,32.82,-137.47,47.88,-110.34],[9E9,9E9,9E9,9E9,9E9,9E9]],speeddata0,DefaultBlend,tool0;
  MoveAbsJ [[-51.46,4.04,32.02,-136.83,47.30,-109.92],[9E9,9E9,9E9,9E9,9E9,9E9]],speeddata0,DefaultBlend,tool0;
  MoveAbsJ [[-50.46,3.76,31.22,-136.19,46.72,-109.49],[9E9,9E9,9E9,9E9,9E9,9E9]],speeddata0,DefaultBlend,tool0;
  MoveAbsJ [[-49.47,3.49,30.42,-135.55,46.15,-109.06],[9E9,9E9,9E9,9E9,9E9,9E9]],speeddata0,DefaultBlend,tool0;
  MoveAbsJ [[-48.47,3.21,29.62,-134.91,45.57,-108.63],[9E9,9E9,9E9,9E9,9E9,9E9]],speeddata0,DefaultBlend,tool0;
  MoveAbsJ [[-47.48,2.94,28.82,-134.27,45.00,-108.21],[9E9,9E9,9E9,9E9,9E9,9E9]],speeddata0,DefaultBlend,tool0;
  MoveAbsJ [[-46.48,2.66,28.02,-133.63,44.42,-107.78],[9E9,9E9,9E9,9E9,9E9,9E9]],speeddata0,DefaultBlend,tool0;
  MoveAbsJ [[-45.49,2.39,27.22,-132.99,43.84,-107.35],[9E9,9E9,9E9,9E9,9E9,9E9]],speeddata0,DefaultBlend,tool0;
  MoveAbsJ [[-44.49,2.12,26.41,-132.35,43.27,-106.92],[9E9,9E9,9E9,9E9,9E9,9E9]],speeddata0,DefaultBlend,tool0;
  MoveAbsJ [[-43.50,1.84,25.61,-131.71,42.69,-106.50],[9E9,9E9,9E9,9E9,9E9,9E9]],speeddata0,DefaultBlend,tool0;
  MoveAbsJ [[-42.50,1.57,24.81,-131.07,42.12,-106.07],[9E9,9E9,9E9,9E9,9E9,9E9]],speeddata0,DefaultBlend,tool0;
  MoveAbsJ [[-41.51,1.29,24.01,-130.43,41.54,-105.64],[9E9,9E9,9E9,9E9,9E9,9E9]],speeddata0,DefaultBlend,tool0;
  MoveAbsJ [[-40.51,1.02,23.21,-129.79,40.97,-105.21],[9E9,9E9,9E9,9E9,9E9,9E9]],speeddata0,DefaultBlend,tool0;
  MoveAbsJ [[-39.51,0.74,22.41,-129.16,40.39,-104.79],[9E9,9E9,9E9,9E9,9E9,9E9]],speeddata0,DefaultBlend,tool0;
  MoveAbsJ [[-38.52,0.47,21.61,-128.52,39.81,-104.36],[9E9,9E9,9E9,9E9,9E9,9E9]],speeddata0,DefaultBlend,tool0;
  MoveAbsJ [[-37.52,0.20,20.81,-127.88,39.24,-103.93],[9E9,9E9,9E9,9E9,9E9,9E9]],speeddata0,DefaultBlend,tool0;
  MoveAbsJ [[-36.53,-0.08,20.01,-127.24,38.66,-103.50],[9E9,9E9,9E9,9E9,9E9,9E9]],speeddata0,DefaultBlend,tool0;
  MoveAbsJ [[-35.53,-0.35,19.21,-126.60,38.09,-103.08],[9E9,9E9,9E9,9E9,9E9,9E9]],speeddata0,DefaultBlend,tool0;
  MoveAbsJ [[-34.54,-0.63,18.41,-125.96,37.51,-102.65],[9E9,9E9,9E9,9E9,9E9,9E9]],speeddata0,DefaultBlend,tool0;
  MoveAbsJ [[-33.54,-0.90,17.60,-125.32,36.93,-102.22],[9E9,9E9,9E9,9E9,9E9,9E9]],speeddata0,DefaultBlend,tool0;
  MoveAbsJ [[-32.55,-1.18,16.80,-124.68,36.36,-101.80],[9E9,9E9,9E9,9E9,9E9,9E9]],speeddata0,DefaultBlend,tool0;
  MoveAbsJ [[-31.55,-1.45,16.00,-124.04,35.78,-101.37],[9E9,9E9,9E9,9E9,9E9,9E9]],speeddata0,DefaultBlend,tool0;
  MoveAbsJ [[-30.56,-1.72,15.20,-123.40,35.21,-100.94],[9E9,9E9,9E9,9E9,9E9,9E9]],speeddata0,DefaultBlend,tool0;
  MoveAbsJ [[-29.56,-2.00,14.40,-122.76,34.63,-100.51],[9E9,9E9,9E9,9E9,9E9,9E9]],speeddata0,DefaultBlend,tool0;
  MoveAbsJ [[-28.56,-2.27,13.60,-122.12,34.05,-100.09],[9E9,9E9,9E9,9E9,9E9,9E9]],speeddata0,DefaultBlend,tool0;
  MoveAbsJ [[-27.57,-2.55,12.80,-121.48,33.48,-99.66],[9E9,9E9,9E9,9E9,9E9,9E9]],speeddata0,DefaultBlend,tool0;
  MoveAbsJ [[-26.57,-2.82,12.00,-120.84,32.90,-99.23],[9E9,9E9,9E9,9E9,9E9,9E9]],speeddata0,DefaultBlend,tool0;
  MoveAbsJ [[-25.58,-3.10,11.20,-120.20,32.33,-98.80],[9E9,9E9,9E9,9E9,9E9,9E9]],speeddata0,DefaultBlend,tool0;
  MoveAbsJ [[-24.58,-3.37,10.40,-119.56,31.75,-98.38],[9E9,9E9,9E9,9E9,9E9,9E9]],speeddata0,DefaultBlend,tool0;
  MoveAbsJ [[-23.59,-3.64,9.59,-118.93,31.17,-97.95],[9E9,9E9,9E9,9E9,9E9,9E9]],speeddata0,DefaultBlend,tool0;
  MoveAbsJ [[-22.59,-3.92,8.79,-118.29,30.60,-97.52],[9E9,9E9,9E9,9E9,9E9,9E9]],speeddata0,DefaultBlend,tool0;
  MoveAbsJ [[-21.60,-4.19,7.99,-117.65,30.02,-97.09],[9E9,9E9,9E9,9E9,9E9,9E9]],speeddata0,DefaultBlend,tool0;
  MoveAbsJ [[-20.60,-4.47,7.19,-117.01,29.45,-96.67],[9E9,9E9,9E9,9E9,9E9,9E9]],speeddata0,DefaultBlend,tool0;
  MoveAbsJ [[-19.61,-4.74,6.39,-116.37,28.87,-96.24],[9E9,9E9,9E9,9E9,9E9,9E9]],speeddata0,DefaultBlend,tool0;
  MoveAbsJ [[-18.61,-5.02,5.59,-115.73,28.29,-95.81],[9E9,9E9,9E9,9E9,9E9,9E9]],speeddata0,DefaultBlend,tool0;
  MoveAbsJ [[-17.61,-5.29,4.79,-115.09,27.72,-95.38],[9E9,9E9,9E9,9E9,9E9,9E9]],speeddata0,DefaultBlend,tool0;
  MoveAbsJ [[-16.62,-5.56,3.99,-114.45,27.14,-94.96],[9E9,9E9,9E9,9E9,9E9,9E9]],speeddata0,DefaultBlend,tool0;
  MoveAbsJ [[-15.62,-5.84,3.19,-113.81,26.57,-94.53],[9E9,9E9,9E9,9E9,9E9,9E9]],speeddata0,DefaultBlend,tool0;
  MoveAbsJ [[-14.63,-6.11,2.39,-113.17,25.99,-94.10],[9E9,9E9,9E9,9E9,9E9,9E9]],speeddata0,DefaultBlend,tool0;
  MoveAbsJ [[-13.63,-6.39,1.58,-112.53,25.42,-93.67],[9E9,9E9,9E9,9E9,9E9,9E9]],speeddata0,DefaultBlend,tool0;
  MoveAbsJ [[-12.64,-6.66,0.78,-111.89,24.84,-93.25],[9E9,9E9,9E9,9E9,9E9,9E9]],speeddata0,DefaultBlend,tool0;
  MoveAbsJ [[-11.64,-6.94,-0.02,-111.25,24.26,-92.82],[9E9,9E9,9E9,9E9,9E9,9E9]],speeddata0,DefaultBlend,tool0;
  MoveAbsJ [[-10.65,-7.21,-0.82,-110.61,23.69,-92.39],[9E9,9E9,9E9,9E9,9E9,9E9]],speeddata0,DefaultBlend,tool0;
  MoveAbsJ [[-9.65,-7.48,-1.62,-109.97,23.11,-91.96],[9E9,9E9,9E9,9E9,9E9,9E9]],speeddata0,DefaultBlend,tool0;
  MoveAbsJ [[-8.66,-7.76,-2.42,-109.33,22.54,-91.54],[9E9,9E9,9E9,9E9,9E9,9E9]],speeddata0,DefaultBlend,tool0;
  MoveAbsJ [[-7.66,-8.03,-3.22,-108.70,21.96,-91.11],[9E9,9E9,9E9,9E9,9E9,9E9]],speeddata0,DefaultBlend,tool0;
  MoveAbsJ [[-6.66,-8.31,-4.02,-108.06,21.38,-90.68],[9E9,9E9,9E9,9E9,9E9,9E9]],speeddata0,DefaultBlend,tool0;
  MoveAbsJ [[-5.67,-8.58,-4.82,-107.42,20.81,-90.25],[9E9,9E9,9E9,9E9,9E9,9E9]],speeddata0,DefaultBlend,tool0;
  MoveAbsJ [[-4.67,-8.86,-5.62,-106.78,20.23,-89.83],[9E9,9E9,9E9,9E9,9E9,9E9]],speeddata0,DefaultBlend,tool0;
  MoveAbsJ [[-3.68,-9.13,-6.43,-106.14,19.66,-89.40],[9E9,9E9,9E9,9E9,9E9,9E9]],speeddata0,DefaultBlend,tool0;
  MoveAbsJ [[-2.68,-9.40,-7.23,-105.50,19.08,-88.97],[9E9,9E9,9E9,9E9,9E9,9E9]],speeddata0,DefaultBlend,tool0;
  MoveAbsJ [[-1.69,-9.68,-8.03,-104.86,18.50,-88.54],[9E9,9E9,9E9,9E9,9E9,9E9]],speeddata0,DefaultBlend,tool0;
  MoveAbsJ [[-0.69,-9.95,-8.83,-104.22,17.93,-88.12],[9E9,9E9,9E9,9E9,9E9,9E9]],speeddata0,DefaultBlend,tool0;
  MoveAbsJ [[0.30,-10.23,-9.63,-103.58,17.35,-87.69],[9E9,9E9,9E9,9E9,9E9,9E9]],speeddata0,DefaultBlend,tool0;
  MoveAbsJ [[1.30,-10.50,-10.43,-102.94,16.78,-87.26],[9E9,9E9,9E9,9E9,9E9,9E9]],speeddata0,DefaultBlend,tool0;
  MoveAbsJ [[2.29,-10.78,-11.23,-102.30,16.20,-86.83],[9E9,9E9,9E9,9E9,9E9,9E9]],speeddata0,DefaultBlend,tool0;
  MoveAbsJ [[3.29,-11.05,-12.03,-101.66,15.62,-86.41],[9E9,9E9,9E9,9E9,9E9,9E9]],speeddata0,DefaultBlend,tool0;
  MoveAbsJ [[4.28,-11.32,-12.83,-101.02,15.05,-85.98],[9E9,9E9,9E9,9E9,9E9,9E9]],speeddata0,DefaultBlend,tool0;
  MoveAbsJ [[5.28,-11.60,-13.63,-100.38,14.47,-85.55],[9E9,9E9,9E9,9E9,9E9,9E9]],speeddata0,DefaultBlend,tool0;
  MoveAbsJ [[6.28,-11.87,-14.44,-99.74,13.90,-85.12],[9E9,9E9,9E9,9E9,9E9,9E9]],speeddata0,DefaultBlend,tool0;
  MoveAbsJ [[7.27,-12.15,-15.24,-99.10,13.32,-84.70],[9E9,9E9,9E9,9E9,9E9,9E9]],speeddata0,DefaultBlend,tool0;
  MoveAbsJ [[8.27,-12.42,-16.04,-98.47,12.74,-84.27],[9E9,9E9,9E9,9E9,9E9,9E9]],speeddata0,DefaultBlend,tool0;
  MoveAbsJ [[9.26,-12.70,-16.84,-97.83,12.17,-83.84],[9E9,9E9,9E9,9E9,9E9,9E9]],speeddata0,DefaultBlend,tool0;
  MoveAbsJ [[10.26,-12.97,-17.64,-97.19,11.59,-83.41],[9E9,9E9,9E9,9E9,9E9,9E9]],speeddata0,DefaultBlend,tool0;
  MoveAbsJ [[11.25,-13.24,-18.44,-96.55,11.02,-82.99],[9E9,9E9,9E9,9E9,9E9,9E9]],speeddata0,DefaultBlend,tool0;
  MoveAbsJ [[12.25,-13.52,-19.24,-95.91,10.44,-82.56],[9E9,9E9,9E9,9E9,9E9,9E9]],speeddata0,DefaultBlend,tool0;
  MoveAbsJ [[13.24,-13.79,-20.04,-95.27,9.87,-82.13],[9E9,9E9,9E9,9E9,9E9,9E9]],speeddata0,DefaultBlend,tool0;
  MoveAbsJ [[14.24,-14.07,-20.84,-94.63,9.29,-81.70],[9E9,9E9,9E9,9E9,9E9,9E9]],speeddata0,DefaultBlend,tool0;
  MoveAbsJ [[15.23,-14.34,-21.64,-93.99,8.71,-81.28],[9E9,9E9,9E9,9E9,9E9,9E9]],speeddata0,DefaultBlend,tool0;
  MoveAbsJ [[16.23,-14.62,-22.45,-93.35,8.14,-80.85],[9E9,9E9,9E9,9E9,9E9,9E9]],speeddata0,DefaultBlend,tool0;
  MoveAbsJ [[17.23,-14.89,-23.25,-92.71,7.56,-80.42],[9E9,9E9,9E9,9E9,9E9,9E9]],speeddata0,DefaultBlend,tool0;
  MoveAbsJ [[18.22,-15.16,-24.05,-92.07,6.99,-79.99],[9E9,9E9,9E9,9E9,9E9,9E9]],speeddata0,DefaultBlend,tool0;
  MoveAbsJ [[19.22,-15.44,-24.85,-91.43,6.41,-79.57],[9E9,9E9,9E9,9E9,9E9,9E9]],speeddata0,DefaultBlend,tool0;
  MoveAbsJ [[20.21,-15.71,-25.65,-90.79,5.83,-79.14],[9E9,9E9,9E9,9E9,9E9,9E9]],speeddata0,DefaultBlend,tool0;
  MoveAbsJ [[21.21,-15.99,-26.45,-90.15,5.26,-78.71],[9E9,9E9,9E9,9E9,9E9,9E9]],speeddata0,DefaultBlend,tool0;
  MoveAbsJ [[22.20,-16.26,-27.25,-89.51,4.68,-78.28],[9E9,9E9,9E9,9E9,9E9,9E9]],speeddata0,DefaultBlend,tool0;
  MoveAbsJ [[23.20,-16.54,-28.05,-88.87,4.11,-77.86],[9E9,9E9,9E9,9E9,9E9,9E9]],speeddata0,DefaultBlend,tool0;
  MoveAbsJ [[24.19,-16.81,-28.85,-88.23,3.53,-77.43],[9E9,9E9,9E9,9E9,9E9,9E9]],speeddata0,DefaultBlend,tool0;
  MoveAbsJ [[25.19,-17.08,-29.65,-87.60,2.95,-77.00],[9E9,9E9,9E9,9E9,9E9,9E9]],speeddata0,DefaultBlend,tool0;
  MoveAbsJ [[26.18,-17.36,-30.46,-86.96,2.38,-76.57],[9E9,9E9,9E9,9E9,9E9,9E9]],speeddata0,DefaultBlend,tool0;
  MoveAbsJ [[27.18,-17.63,-31.26,-86.32,1.80,-76.15],[9E9,9E9,9E9,9E9,9E9,9E9]],speeddata0,DefaultBlend,tool0;
  MoveAbsJ [[28.18,-17.91,-32.06,-85.68,1.23,-75.72],[9E9,9E9,9E9,9E9,9E9,9E9]],speeddata0,DefaultBlend,tool0;
  MoveAbsJ [[29.17,-18.18,-32.86,-85.04,0.65,-75.29],[9E9,9E9,9E9,9E9,9E9,9E9]],speeddata0,DefaultBlend,tool0;
  MoveAbsJ [[30.17,-18.46,-33.66,-84.40,0.07,-74.86],[9E9,9E9,9E9,9E9,9E9,9E9]],speeddata0,DefaultBlend,tool0;
  MoveAbsJ [[31.16,-18.73,-34.46,-83.76,-0.50,-74.44],[9E9,9E9,9E9,9E9,9E9,9E9]],speeddata0,DefaultBlend,tool0;
  MoveAbsJ [[32.16,-19.00,-35.26,-83.12,-1.08,-74.01],[9E9,9E9,9E9,9E9,9E9,9E9]],speeddata0,DefaultBlend,tool0;
  MoveAbsJ [[33.15,-19.28,-36.06,-82.48,-1.65,-73.58],[9E9,9E9,9E9,9E9,9E9,9E9]],speeddata0,DefaultBlend,tool0;
  MoveAbsJ [[34.15,-19.55,-36.86,-81.84,-2.23,-73.15],[9E9,9E9,9E9,9E9,9E9,9E9]],speeddata0,DefaultBlend,tool0;
  MoveAbsJ [[35.14,-19.83,-37.66,-81.20,-2.81,-72.73],[9E9,9E9,9E9,9E9,9E9,9E9]],speeddata0,DefaultBlend,tool0;
  MoveAbsJ [[36.14,-20.10,-38.47,-80.56,-3.38,-72.30],[9E9,9E9,9E9,9E9,9E9,9E9]],speeddata0,DefaultBlend,tool0;
  MoveAbsJ [[37.13,-20.38,-39.27,-79.92,-3.96,-71.87],[9E9,9E9,9E9,9E9,9E9,9E9]],speeddata0,DefaultBlend,tool0;
  MoveAbsJ [[38.13,-20.65,-40.07,-79.28,-4.53,-71.44],[9E9,9E9,9E9,9E9,9E9,9E9]],speeddata0,DefaultBlend,tool0;
  MoveAbsJ [[39.13,-20.92,-40.87,-78.64,-5.11,-71.02],[9E9,9E9,9E9,9E9,9E9,9E9]],speeddata0,DefaultBlend,tool0;
  MoveAbsJ [[40.12,-21.20,-41.67,-78.00,-5.69,-70.59],[9E9,9E9,9E9,9E9,9E9,9E9]],speeddata0,DefaultBlend,tool0;
  MoveAbsJ [[41.12,-21.47,-42.47,-77.37,-6.26,-70.16],[9E9,9E9,9E9,9E9,9E9,9E9]],speeddata0,DefaultBlend,tool0;
  MoveAbsJ [[42.11,-21.75,-43.27,-76.73,-6.84,-69.73],[9E9,9E9,9E9,9E9,9E9,9E9]],speeddata0,DefaultBlend,tool0;
  MoveAbsJ [[43.11,-22.02,-44.07,-76.09,-7.41,-69.31],[9E9,9E9,9E9,9E9,9E9,9E9]],speeddata0,DefaultBlend,tool0;
  MoveAbsJ [[44.10,-22.30,-44.87,-75.45,-7.99,-68.88],[9E9,9E9,9E9,9E9,9E9,9E9]],speeddata0,DefaultBlend,tool0;
  MoveAbsJ [[45.10,-22.57,-45.67,-74.81,-8.56,-68.45],[9E9,9E9,9E9,9E9,9E9,9E9]],speeddata0,DefaultBlend,tool0;
  MoveAbsJ [[46.09,-22.84,-46.48,-74.17,-9.14,-68.02],[9E9,9E9,9E9,9E9,9E9,9E9]],speeddata0,DefaultBlend,tool0;
  MoveAbsJ [[47.09,-23.12,-47.28,-73.53,-9.72,-67.60],[9E9,9E9,9E9,9E9,9E9,9E9]],speeddata0,DefaultBlend,tool0;
  MoveAbsJ [[48.08,-23.39,-48.08,-72.89,-10.29,-67.17],[9E9,9E9,9E9,9E9,9E9,9E9]],speeddata0,DefaultBlend,tool0;
  MoveAbsJ [[49.08,-23.67,-48.88,-72.25,-10.87,-66.74],[9E9,9E9,9E9,9E9,9E9,9E9]],speeddata0,DefaultBlend,tool0;
  MoveAbsJ [[50.08,-23.94,-49.68,-71.61,-11.44,-66.31],[9E9,9E9,9E9,9E9,9E9,9E9]],speeddata0,DefaultBlend,tool0;
  MoveAbsJ [[51.07,-24.22,-50.48,-70.97,-12.02,-65.89],[9E9,9E9,9E9,9E9,9E9,9E9]],speeddata0,DefaultBlend,tool0;
  MoveAbsJ [[52.07,-24.49,-51.28,-70.33,-12.60,-65.46],[9E9,9E9,9E9,9E9,9E9,9E9]],speeddata0,DefaultBlend,tool0;
  MoveAbsJ [[53.06,-24.76,-52.08,-69.69,-13.17,-65.03],[9E9,9E9,9E9,9E9,9E9,9E9]],speeddata0,DefaultBlend,tool0;
  MoveAbsJ [[54.06,-25.04,-52.88,-69.05,-13.75,-64.60],[9E9,9E9,9E9,9E9,9E9,9E9]],speeddata0,DefaultBlend,tool0;
  MoveAbsJ [[55.05,-25.31,-53.68,-68.41,-14.32,-64.18],[9E9,9E9,9E9,9E9,9E9,9E9]],speeddata0,DefaultBlend,tool0;
  MoveAbsJ [[56.05,-25.59,-54.48,-67.77,-14.90,-63.75],[9E9,9E9,9E9,9E9,9E9,9E9]],speeddata0,DefaultBlend,tool0;
  MoveAbsJ [[57.04,-25.86,-55.29,-67.14,-15.48,-63.32],[9E9,9E9,9E9,9E9,9E9,9E9]],speeddata0,DefaultBlend,tool0;
  MoveAbsJ [[58.04,-26.14,-56.09,-66.50,-16.05,-62.89],[9E9,9E9,9E9,9E9,9E9,9E9]],speeddata0,DefaultBlend,tool0;
  MoveAbsJ [[59.03,-26.41,-56.89,-65.86,-16.63,-62.47],[9E9,9E9,9E9,9E9,9E9,9E9]],speeddata0,DefaultBlend,tool0;
  MoveAbsJ [[60.03,-26.68,-57.69,-65.22,-17.20,-62.04],[9E9,9E9,9E9,9E9,9E9,9E9]],speeddata0,DefaultBlend,tool0;
  MoveAbsJ [[61.03,-26.96,-58.49,-64.58,-17.78,-61.61],[9E9,9E9,9E9,9E9,9E9,9E9]],speeddata0,DefaultBlend,tool0;
  MoveAbsJ [[62.02,-27.23,-59.29,-63.94,-18.36,-61.18],[9E9,9E9,9E9,9E9,9E9,9E9]],speeddata0,DefaultBlend,tool0;
  MoveAbsJ [[63.02,-27.51,-60.09,-63.30,-18.93,-60.76],[9E9,9E9,9E9,9E9,9E9,9E9]],speeddata0,DefaultBlend,tool0;
  MoveAbsJ [[64.01,-27.78,-60.89,-62.66,-19.51,-60.33],[9E9,9E9,9E9,9E9,9E9,9E9]],speeddata0,DefaultBlend,tool0;
  MoveAbsJ [[65.01,-28.06,-61.69,-62.02,-20.08,-59.90],[9E9,9E9,9E9,9E9,9E9,9E9]],speeddata0,DefaultBlend,tool0;
  MoveAbsJ [[66.00,-28.33,-62.49,-61.38,-20.66,-59.47],[9E9,9E9,9E9,9E9,9E9,9E9]],speeddata0,DefaultBlend,tool0;
  MoveAbsJ [[67.00,-28.60,-63.30,-60.74,-21.24,-59.05],[9E9,9E9,9E9,9E9,9E9,9E9]],speeddata0,DefaultBlend,tool0;
  MoveAbsJ [[67.99,-28.88,-64.10,-60.10,-21.81,-58.62],[9E9,9E9,9E9,9E9,9E9,9E9]],speeddata0,DefaultBlend,tool0;
  MoveAbsJ [[68.99,-29.15,-64.90,-59.46,-22.39,-58.19],[9E9,9E9,9E9,9E9,9E9,9E9]],speeddata0,DefaultBlend,tool0;
  MoveAbsJ [[69.98,-29.43,-65.70,-58.82,-22.96,-57.76],[9E9,9E9,9E9,9E9,9E9,9E9]],speeddata0,DefaultBlend,tool0;
  MoveAbsJ [[70.98,-29.70,-66.50,-58.18,-23.54,-57.34],[9E9,9E9,9E9,9E9,9E9,9E9]],speeddata0,DefaultBlend,tool0;
  MoveAbsJ [[71.98,-29.98,-67.30,-57.54,-24.11,-56.91],[9E9,9E9,9E9,9E9,9E9,9E9]],speeddata0,DefaultBlend,tool0;
  MoveAbsJ [[72.97,-30.25,-68.10,-56.91,-24.69,-56.48],[9E9,9E9,9E9,9E9,9E9,9E9]],speeddata0,DefaultBlend,tool0;
  MoveAbsJ [[73.97,-30.52,-68.90,-56.27,-25.27,-56.05],[9E9,9E9,9E9,9E9,9E9,9E9]],speeddata0,DefaultBlend,tool0;
  MoveAbsJ [[74.96,-30.80,-69.70,-55.63,-25.84,-55.63],[9E9,9E9,9E9,9E9,9E9,9E9]],speeddata0,DefaultBlend,tool0;
  MoveAbsJ [[75.96,-31.07,-70.50,-54.99,-26.42,-55.20],[9E9,9E9,9E9,9E9,9E9,9E9]],speeddata0,DefaultBlend,tool0;
  MoveAbsJ [[76.95,-31.35,-71.31,-54.35,-26.99,-54.77],[9E9,9E9,9E9,9E9,9E9,9E9]],speeddata0,DefaultBlend,tool0;
  MoveAbsJ [[77.95,-31.62,-72.11,-53.71,-27.57,-54.34],[9E9,9E9,9E9,9E9,9E9,9E9]],speeddata0,DefaultBlend,tool0;
  MoveAbsJ [[78.94,-31.90,-72.91,-53.07,-28.15,-53.92],[9E9,9E9,9E9,9E9,9E9,9E9]],speeddata0,DefaultBlend,tool0;
  MoveAbsJ [[79.94,-32.17,-73.71,-52.43,-28.72,-53.49],[9E9,9E9,9E9,9E9,9E9,9E9]],speeddata0,DefaultBlend,tool0;
  MoveAbsJ [[80.93,-32.44,-74.51,-51.79,-29.30,-53.06],[9E9,9E9,9E9,9E9,9E9,9E9]],speeddata0,DefaultBlend,tool0;
  MoveAbsJ [[81.93,-32.72,-75.31,-51.15,-29.87,-52.63],[9E9,9E9,9E9,9E9,9E9,9E9]],speeddata0,DefaultBlend,tool0;
  MoveAbsJ [[82.92,-32.99,-76.11,-50.51,-30.45,-52.21],[9E9,9E9,9E9,9E9,9E9,9E9]],speeddata0,DefaultBlend,tool0;
  MoveAbsJ [[83.92,-33.27,-76.91,-49.87,-31.03,-51.78],[9E9,9E9,9E9,9E9,9E9,9E9]],speeddata0,DefaultBlend,tool0;
  MoveAbsJ [[84.92,-33.54,-77.71,-49.23,-31.60,-51.35],[9E9,9E9,9E9,9E9,9E9,9E9]],speeddata0,DefaultBlend,tool0;
  MoveAbsJ [[85.91,-33.82,-78.51,-48.59,-32.18,-50.92],[9E9,9E9,9E9,9E9,9E9,9E9]],speeddata0,DefaultBlend,tool0;
  MoveAbsJ [[86.91,-34.09,-79.32,-47.95,-32.75,-50.50],[9E9,9E9,9E9,9E9,9E9,9E9]],speeddata0,DefaultBlend,tool0;
  MoveAbsJ [[87.90,-34.36,-80.12,-47.31,-33.33,-50.07],[9E9,9E9,9E9,9E9,9E9,9E9]],speeddata0,DefaultBlend,tool0;
  MoveAbsJ [[88.90,-34.64,-80.92,-46.68,-33.91,-49.64],[9E9,9E9,9E9,9E9,9E9,9E9]],speeddata0,DefaultBlend,tool0;
  MoveAbsJ [[89.89,-34.91,-81.72,-46.04,-34.48,-49.21],[9E9,9E9,9E9,9E9,9E9,9E9]],speeddata0,DefaultBlend,tool0;
  MoveAbsJ [[90.89,-35.19,-82.52,-45.40,-35.06,-48.79],[9E9,9E9,9E9,9E9,9E9,9E9]],speeddata0,DefaultBlend,tool0;
  MoveAbsJ [[91.88,-35.46,-83.32,-44.76,-35.63,-48.36],[9E9,9E9,9E9,9E9,9E9,9E9]],speeddata0,DefaultBlend,tool0;
  MoveAbsJ [[92.88,-35.74,-84.12,-44.12,-36.21,-47.93],[9E9,9E9,9E9,9E9,9E9,9E9]],speeddata0,DefaultBlend,tool0;
  MoveAbsJ [[93.87,-36.01,-84.92,-43.48,-36.79,-47.50],[9E9,9E9,9E9,9E9,9E9,9E9]],speeddata0,DefaultBlend,tool0;
  MoveAbsJ [[94.87,-36.28,-85.72,-42.84,-37.36,-47.08],[9E9,9E9,9E9,9E9,9E9,9E9]],speeddata0,DefaultBlend,tool0;
  MoveAbsJ [[95.87,-36.56,-86.52,-42.20,-37.94,-46.65],[9E9,9E9,9E9,9E9,9E9,9E9]],speeddata0,DefaultBlend,tool0;
  MoveAbsJ [[96.86,-36.83,-87.33,-41.56,-38.51,-46.22],[9E9,9E9,9E9,9E9,9E9,9E9]],speeddata0,DefaultBlend,tool0;
  MoveAbsJ [[97.86,-37.11,-88.13,-40.92,-39.09,-45.79],[9E9,9E9,9E9,9E9,9E9,9E9]],speeddata0,DefaultBlend,tool0;
  MoveAbsJ [[98.85,-37.38,-88.93,-40.28,-39.66,-45.37],[9E9,9E9,9E9,9E9,9E9,9E9]],speeddata0,DefaultBlend,tool0;
  MoveAbsJ [[99.85,-37.66,-89.73,-39.64,-40.24,-44.94],[9E9,9E9,9E9,9E9,9E9,9E9]],speeddata0,DefaultBlend,tool0;
  MoveAbsJ [[100.84,-37.93,-90.53,-39.00,-40.82,-44.51],[9E9,9E9,9E9,9E9,9E9,9E9]],speeddata0,DefaultBlend,tool0;
  MoveAbsJ [[101.84,-38.20,-91.33,-38.36,-41.39,-44.08],[9E9,9E9,9E9,9E9,9E9,9E9]],speeddata0,DefaultBlend,tool0;
  MoveAbsJ [[102.83,-38.48,-92.13,-37.72,-41.97,-43.66],[9E9,9E9,9E9,9E9,9E9,9E9]],speeddata0,DefaultBlend,tool0;
  MoveAbsJ [[103.83,-38.75,-92.93,-37.08,-42.54,-43.23],[9E9,9E9,9E9,9E9,9E9,9E9]],speeddata0,DefaultBlend,tool0;
  MoveAbsJ [[104.82,-39.03,-93.73,-36.44,-43.12,-42.80],[9E9,9E9,9E9,9E9,9E9,9E9]],speeddata0,DefaultBlend,tool0;
  MoveAbsJ [[105.82,-39.30,-94.53,-35.81,-43.70,-42.37],[9E9,9E9,9E9,9E9,9E9,9E9]],speeddata0,DefaultBlend,tool0;
  MoveAbsJ [[106.82,-39.58,-95.34,-35.17,-44.27,-41.95],[9E9,9E9,9E9,9E9,9E9,9E9]],speeddata0,DefaultBlend,tool0;
  MoveAbsJ [[107.81,-39.85,-96.14,-34.53,-44.85,-41.52],[9E9,9E9,9E9,9E9,9E9,9E9]],speeddata0,DefaultBlend,tool0;
  MoveAbsJ [[108.81,-40.12,-96.94,-33.89,-45.42,-41.09],[9E9,9E9,9E9,9E9,9E9,9E9]],speeddata0,DefaultBlend,tool0;
  MoveAbsJ [[109.80,-40.40,-97.74,-33.25,-46.00,-40.66],[9E9,9E9,9E9,9E9,9E9,9E9]],speeddata0,DefaultBlend,tool0;
  MoveAbsJ [[110.80,-40.67,-98.54,-32.61,-46.58,-40.24],[9E9,9E9,9E9,9E9,9E9,9E9]],speeddata0,DefaultBlend,tool0;
  MoveAbsJ [[111.79,-40.95,-99.34,-31.97,-47.15,-39.81],[9E9,9E9,9E9,9E9,9E9,9E9]],speeddata0,DefaultBlend,tool0;
  MoveAbsJ [[112.79,-41.22,-100.14,-31.33,-47.73,-39.38],[9E9,9E9,9E9,9E9,9E9,9E9]],speeddata0,DefaultBlend,tool0;
  MoveAbsJ [[113.78,-41.50,-100.94,-30.69,-48.30,-38.95],[9E9,9E9,9E9,9E9,9E9,9E9]],speeddata0,DefaultBlend,tool0;
  MoveAbsJ [[114.78,-41.77,-101.74,-30.05,-48.88,-38.53],[9E9,9E9,9E9,9E9,9E9,9E9]],speeddata0,DefaultBlend,tool0;
  MoveAbsJ [[115.77,-42.04,-102.54,-29.41,-49.46,-38.10],[9E9,9E9,9E9,9E9,9E9,9E9]],speeddata0,DefaultBlend,tool0;
  MoveAbsJ [[116.77,-42.32,-103.35,-28.77,-50.03,-37.67],[9E9,9E9,9E9,9E9,9E9,9E9]],speeddata0,DefaultBlend,tool0;
  MoveAbsJ [[117.77,-42.59,-104.15,-28.13,-50.61,-37.24],[9E9,9E9,9E9,9E9,9E9,9E9]],speeddata0,DefaultBlend,tool0;
  MoveAbsJ [[118.76,-42.87,-104.95,-27.49,-51.18,-36.82],[9E9,9E9,9E9,9E9,9E9,9E9]],speeddata0,DefaultBlend,tool0;
  MoveAbsJ [[119.76,-43.14,-105.75,-26.85,-51.76,-36.39],[9E9,9E9,9E9,9E9,9E9,9E9]],speeddata0,DefaultBlend,tool0;
  MoveAbsJ [[120.75,-43.42,-106.55,-26.21,-52.34,-35.96],[9E9,9E9,9E9,9E9,9E9,9E9]],speeddata0,DefaultBlend,tool0;
  MoveAbsJ [[121.75,-43.69,-107.35,-25.58,-52.91,-35.53],[9E9,9E9,9E9,9E9,9E9,9E9]],speeddata0,DefaultBlend,tool0;
  MoveAbsJ [[122.74,-43.96,-108.15,-24.94,-53.49,-35.11],[9E9,9E9,9E9,9E9,9E9,9E9]],speeddata0,DefaultBlend,tool0;
  MoveAbsJ [[123.74,-44.24,-108.95,-24.30,-54.06,-34.68],[9E9,9E9,9E9,9E9,9E9,9E9]],speeddata0,DefaultBlend,tool0;
  MoveAbsJ [[124.73,-44.51,-109.75,-23.66,-54.64,-34.25],[9E9,9E9,9E9,9E9,9E9,9E9]],speeddata0,DefaultBlend,tool0;
  MoveAbsJ [[125.73,-44.79,-110.55,-23.02,-55.21,-33.82],[9E9,9E9,9E9,9E9,9E9,9E9]],speeddata0,DefaultBlend,tool0;
  MoveAbsJ [[126.72,-45.06,-111.36,-22.38,-55.79,-33.40],[9E9,9E9,9E9,9E9,9E9,9E9]],speeddata0,DefaultBlend,tool0;
  MoveAbsJ [[127.72,-45.34,-112.16,-21.74,-56.37,-32.97],[9E9,9E9,9E9,9E9,9E9,9E9]],speeddata0,DefaultBlend,tool0;
  MoveAbsJ [[128.72,-45.61,-112.96,-21.10,-56.94,-32.54],[9E9,9E9,9E9,9E9,9E9,9E9]],speeddata0,DefaultBlend,tool0;
  MoveAbsJ [[129.71,-45.88,-113.76,-20.46,-57.52,-32.11],[9E9,9E9,9E9,9E9,9E9,9E9]],speeddata0,DefaultBlend,tool0;
  MoveAbsJ [[130.71,-46.16,-114.56,-19.82,-58.09,-31.69],[9E9,9E9,9E9,9E9,9E9,9E9]],speeddata0,DefaultBlend,tool0;
  MoveAbsJ [[131.70,-46.43,-115.36,-19.18,-58.67,-31.26],[9E9,9E9,9E9,9E9,9E9,9E9]],speeddata0,DefaultBlend,tool0;
  MoveAbsJ [[132.70,-46.71,-116.16,-18.54,-59.25,-30.83],[9E9,9E9,9E9,9E9,9E9,9E9]],speeddata0,DefaultBlend,tool0;
  MoveAbsJ [[133.69,-46.98,-116.96,-17.90,-59.82,-30.40],[9E9,9E9,9E9,9E9,9E9,9E9]],speeddata0,DefaultBlend,tool0;
  MoveAbsJ [[134.69,-47.26,-117.76,-17.26,-60.40,-29.98],[9E9,9E9,9E9,9E9,9E9,9E9]],speeddata0,DefaultBlend,tool0;
  MoveAbsJ [[135.68,-47.53,-118.56,-16.62,-60.97,-29.55],[9E9,9E9,9E9,9E9,9E9,9E9]],speeddata0,DefaultBlend,tool0;
  MoveAbsJ [[136.68,-47.80,-119.36,-15.98,-61.55,-29.12],[9E9,9E9,9E9,9E9,9E9,9E9]],speeddata0,DefaultBlend,tool0;
  MoveAbsJ [[137.67,-48.08,-120.17,-15.35,-62.13,-28.69],[9E9,9E9,9E9,9E9,9E9,9E9]],speeddata0,DefaultBlend,tool0;
  MoveAbsJ [[138.67,-48.35,-120.97,-14.71,-62.70,-28.27],[9E9,9E9,9E9,9E9,9E9,9E9]],speeddata0,DefaultBlend,tool0;
  MoveAbsJ [[139.67,-48.63,-121.77,-14.07,-63.28,-27.84],[9E9,9E9,9E9,9E9,9E9,9E9]],speeddata0,DefaultBlend,tool0;
  MoveAbsJ [[140.66,-48.90,-122.57,-13.43,-63.85,-27.41],[9E9,9E9,9E9,9E9,9E9,9E9]],speeddata0,DefaultBlend,tool0;
  MoveAbsJ [[141.66,-49.18,-123.37,-12.79,-64.43,-26.98],[9E9,9E9,9E9,9E9,9E9,9E9]],speeddata0,DefaultBlend,tool0;
  MoveAbsJ [[142.65,-49.45,-124.17,-12.15,-65.01,-26.56],[9E9,9E9,9E9,9E9,9E9,9E9]],speeddata0,DefaultBlend,tool0;
  MoveAbsJ [[143.65,-49.72,-124.97,-11.51,-65.58,-26.13],[9E9,9E9,9E9,9E9,9E9,9E9]],speeddata0,DefaultBlend,tool0;
  MoveAbsJ [[144.64,-50.00,-125.77,-10.87,-66.16,-25.70],[9E9,9E9,9E9,9E9,9E9,9E9]],speeddata0,DefaultBlend,tool0;
  MoveAbsJ [[145.64,-50.27,-126.57,-10.23,-66.73,-25.27],[9E9,9E9,9E9,9E9,9E9,9E9]],speeddata0,DefaultBlend,tool0;
  MoveAbsJ [[146.63,-50.55,-127.37,-9.59,-67.31,-24.85],[9E9,9E9,9E9,9E9,9E9,9E9]],speeddata0,DefaultBlend,tool0;
  MoveAbsJ [[147.63,-50.82,-128.18,-8.95,-67.89,-24.42],[9E9,9E9,9E9,9E9,9E9,9E9]],speeddata0,DefaultBlend,tool0;
  MoveAbsJ [[148.62,-51.10,-128.98,-8.31,-68.46,-23.99],[9E9,9E9,9E9,9E9,9E9,9E9]],speeddata0,DefaultBlend,tool0;
  MoveAbsJ [[149.62,-51.37,-129.78,-7.67,-69.04,-23.56],[9E9,9E9,9E9,9E9,9E9,9E9]],speeddata0,DefaultBlend,tool0;
  MoveAbsJ [[150.62,-51.64,-130.58,-7.03,-69.61,-23.14],[9E9,9E9,9E9,9E9,9E9,9E9]],speeddata0,DefaultBlend,tool0;
  MoveAbsJ [[151.61,-51.92,-131.38,-6.39,-70.19,-22.71],[9E9,9E9,9E9,9E9,9E9,9E9]],speeddata0,DefaultBlend,tool0;
  MoveAbsJ [[152.61,-52.19,-132.18,-5.75,-70.76,-22.28],[9E9,9E9,9E9,9E9,9E9,9E9]],speeddata0,DefaultBlend,tool0;
  MoveAbsJ [[153.60,-52.47,-132.98,-5.12,-71.34,-21.85],[9E9,9E9,9E9,9E9,9E9,9E9]],speeddata0,DefaultBlend,tool0;
  MoveAbsJ [[154.60,-52.74,-133.78,-4.48,-71.92,-21.43],[9E9,9E9,9E9,9E9,9E9,9E9]],speeddata0,DefaultBlend,tool0;
  MoveAbsJ [[155.59,-53.02,-134.58,-3.84,-72.49,-21.00],[9E9,9E9,9E9,9E9,9E9,9E9]],speeddata0,DefaultBlend,tool0;
  MoveAbsJ [[156.59,-53.29,-135.38,-3.20,-73.07,-20.57],[9E9,9E9,9E9,9E9,9E9,9E9]],speeddata0,DefaultBlend,tool0;
  MoveAbsJ [[157.58,-53.56,-136.19,-2.56,-73.64,-20.14],[9E9,9E9,9E9,9E9,9E9,9E9]],speeddata0,DefaultBlend,tool0;
  MoveAbsJ [[158.58,-53.84,-136.99,-1.92,-74.22,-19.72],[9E9,9E9,9E9,9E9,9E9,9E9]],speeddata0,DefaultBlend,tool0;
  MoveAbsJ [[159.57,-54.11,-137.79,-1.28,-74.80,-19.29],[9E9,9E9,9E9,9E9,9E9,9E9]],speeddata0,DefaultBlend,tool0;
  MoveAbsJ [[160.57,-54.39,-138.59,-0.64,-75.37,-18.86],[9E9,9E9,9E9,9E9,9E9,9E9]],speeddata0,DefaultBlend,tool0;
  MoveAbsJ [[161.57,-54.66,-139.39,-0.00,-75.95,-18.43],[9E9,9E9,9E9,9E9,9E9,9E9]],speeddata0,FinePoint,tool0;
  TPWrite "Action 11 LinearMovement.";
  MoveAbsJ [[161.57,-54.66,-139.39,-0.00,-75.95,-18.43],[9E9,9E9,9E9,9E9,9E9,9E9]],speeddata0,DefaultBlend,tool0;
  MoveAbsJ [[161.57,-55.31,-139.44,-0.00,-75.25,-18.43],[9E9,9E9,9E9,9E9,9E9,9E9]],speeddata0,DefaultBlend,tool0;
  MoveAbsJ [[161.57,-55.96,-139.50,-0.00,-74.54,-18.43],[9E9,9E9,9E9,9E9,9E9,9E9]],speeddata0,DefaultBlend,tool0;
  MoveAbsJ [[161.57,-56.62,-139.54,-0.00,-73.85,-18.43],[9E9,9E9,9E9,9E9,9E9,9E9]],speeddata0,DefaultBlend,tool0;
  MoveAbsJ [[161.57,-57.28,-139.56,-0.00,-73.16,-18.43],[9E9,9E9,9E9,9E9,9E9,9E9]],speeddata0,DefaultBlend,tool0;
  MoveAbsJ [[161.57,-57.96,-139.56,-0.00,-72.48,-18.43],[9E9,9E9,9E9,9E9,9E9,9E9]],speeddata0,DefaultBlend,tool0;
  MoveAbsJ [[161.57,-58.66,-139.52,-0.00,-71.82,-18.43],[9E9,9E9,9E9,9E9,9E9,9E9]],speeddata0,DefaultBlend,tool0;
  MoveAbsJ [[161.57,-59.37,-139.46,-0.00,-71.17,-18.43],[9E9,9E9,9E9,9E9,9E9,9E9]],speeddata0,DefaultBlend,tool0;
  MoveAbsJ [[161.57,-60.10,-139.37,-0.00,-70.53,-18.43],[9E9,9E9,9E9,9E9,9E9,9E9]],speeddata0,FinePoint,tool0;
  TPWrite "Action 12 OpenGripper.";
  TPWrite "Press Play to Continue";
  Stop;
  TPWrite "Action 13 LinearMovement.";
  MoveAbsJ [[161.57,-60.10,-139.36,-0.00,-70.54,-18.43],[9E9,9E9,9E9,9E9,9E9,9E9]],speeddata0,DefaultBlend,tool0;
  MoveAbsJ [[161.57,-59.40,-139.41,-0.00,-71.19,-18.43],[9E9,9E9,9E9,9E9,9E9,9E9]],speeddata0,DefaultBlend,tool0;
  MoveAbsJ [[161.57,-58.68,-139.48,-0.00,-71.84,-18.43],[9E9,9E9,9E9,9E9,9E9,9E9]],speeddata0,DefaultBlend,tool0;
  MoveAbsJ [[161.57,-57.98,-139.52,-0.00,-72.49,-18.43],[9E9,9E9,9E9,9E9,9E9,9E9]],speeddata0,DefaultBlend,tool0;
  MoveAbsJ [[161.57,-57.29,-139.54,-0.00,-73.16,-18.43],[9E9,9E9,9E9,9E9,9E9,9E9]],speeddata0,DefaultBlend,tool0;
  MoveAbsJ [[161.57,-56.62,-139.55,-0.00,-73.84,-18.43],[9E9,9E9,9E9,9E9,9E9,9E9]],speeddata0,DefaultBlend,tool0;
  MoveAbsJ [[161.57,-55.95,-139.53,-0.00,-74.52,-18.43],[9E9,9E9,9E9,9E9,9E9,9E9]],speeddata0,DefaultBlend,tool0;
  MoveAbsJ [[161.57,-55.29,-139.48,-0.00,-75.23,-18.43],[9E9,9E9,9E9,9E9,9E9,9E9]],speeddata0,DefaultBlend,tool0;
  MoveAbsJ [[161.57,-54.66,-139.39,-0.00,-75.95,-18.43],[9E9,9E9,9E9,9E9,9E9,9E9]],speeddata0,FinePoint,tool0;
  TPWrite "Action 14 FreeMovement.";
  MoveAbsJ [[161.57,-54.66,-139.39,-0.00,-75.95,-18.43],[9E9,9E9,9E9,9E9,9E9,9E9]],speeddata0,DefaultBlend,tool0;
  MoveAbsJ [[161.30,-54.43,-139.79,-0.99,-75.74,-17.90],[9E9,9E9,9E9,9E9,9E9,9E9]],speeddata0,DefaultBlend,tool0;
  MoveAbsJ [[161.03,-54.19,-140.20,-1.98,-75.54,-17.37],[9E9,9E9,9E9,9E9,9E9,9E9]],speeddata0,DefaultBlend,tool0;
  MoveAbsJ [[160.76,-53.96,-140.60,-2.97,-75.34,-16.84],[9E9,9E9,9E9,9E9,9E9,9E9]],speeddata0,DefaultBlend,tool0;
  MoveAbsJ [[160.50,-53.72,-141.00,-3.96,-75.13,-16.31],[9E9,9E9,9E9,9E9,9E9,9E9]],speeddata0,DefaultBlend,tool0;
  MoveAbsJ [[160.23,-53.49,-141.41,-4.95,-74.93,-15.78],[9E9,9E9,9E9,9E9,9E9,9E9]],speeddata0,DefaultBlend,tool0;
  MoveAbsJ [[159.96,-53.26,-141.81,-5.94,-74.73,-15.25],[9E9,9E9,9E9,9E9,9E9,9E9]],speeddata0,DefaultBlend,tool0;
  MoveAbsJ [[159.70,-53.02,-142.21,-6.93,-74.52,-14.72],[9E9,9E9,9E9,9E9,9E9,9E9]],speeddata0,DefaultBlend,tool0;
  MoveAbsJ [[159.43,-52.79,-142.62,-7.92,-74.32,-14.18],[9E9,9E9,9E9,9E9,9E9,9E9]],speeddata0,DefaultBlend,tool0;
  MoveAbsJ [[159.16,-52.55,-143.02,-8.91,-74.12,-13.65],[9E9,9E9,9E9,9E9,9E9,9E9]],speeddata0,DefaultBlend,tool0;
  MoveAbsJ [[158.90,-52.32,-143.42,-9.90,-73.92,-13.12],[9E9,9E9,9E9,9E9,9E9,9E9]],speeddata0,DefaultBlend,tool0;
  MoveAbsJ [[158.63,-52.08,-143.83,-10.89,-73.71,-12.59],[9E9,9E9,9E9,9E9,9E9,9E9]],speeddata0,DefaultBlend,tool0;
  MoveAbsJ [[158.36,-51.85,-144.23,-11.88,-73.51,-12.06],[9E9,9E9,9E9,9E9,9E9,9E9]],speeddata0,DefaultBlend,tool0;
  MoveAbsJ [[158.09,-51.62,-144.63,-12.87,-73.31,-11.53],[9E9,9E9,9E9,9E9,9E9,9E9]],speeddata0,DefaultBlend,tool0;
  MoveAbsJ [[157.83,-51.38,-145.04,-13.86,-73.10,-11.00],[9E9,9E9,9E9,9E9,9E9,9E9]],speeddata0,DefaultBlend,tool0;
  MoveAbsJ [[157.56,-51.15,-145.44,-14.85,-72.90,-10.47],[9E9,9E9,9E9,9E9,9E9,9E9]],speeddata0,DefaultBlend,tool0;
  MoveAbsJ [[157.29,-50.91,-145.84,-15.84,-72.70,-9.93],[9E9,9E9,9E9,9E9,9E9,9E9]],speeddata0,DefaultBlend,tool0;
  MoveAbsJ [[157.03,-50.68,-146.24,-16.83,-72.49,-9.40],[9E9,9E9,9E9,9E9,9E9,9E9]],speeddata0,DefaultBlend,tool0;
  MoveAbsJ [[156.76,-50.45,-146.65,-17.82,-72.29,-8.87],[9E9,9E9,9E9,9E9,9E9,9E9]],speeddata0,DefaultBlend,tool0;
  MoveAbsJ [[156.49,-50.21,-147.05,-18.81,-72.09,-8.34],[9E9,9E9,9E9,9E9,9E9,9E9]],speeddata0,DefaultBlend,tool0;
  MoveAbsJ [[156.23,-49.98,-147.45,-19.80,-71.88,-7.81],[9E9,9E9,9E9,9E9,9E9,9E9]],speeddata0,DefaultBlend,tool0;
  MoveAbsJ [[155.96,-49.74,-147.86,-20.79,-71.68,-7.28],[9E9,9E9,9E9,9E9,9E9,9E9]],speeddata0,DefaultBlend,tool0;
  MoveAbsJ [[155.69,-49.51,-148.26,-21.78,-71.48,-6.75],[9E9,9E9,9E9,9E9,9E9,9E9]],speeddata0,DefaultBlend,tool0;
  MoveAbsJ [[155.42,-49.27,-148.66,-22.77,-71.27,-6.21],[9E9,9E9,9E9,9E9,9E9,9E9]],speeddata0,DefaultBlend,tool0;
  MoveAbsJ [[155.16,-49.04,-149.07,-23.76,-71.07,-5.68],[9E9,9E9,9E9,9E9,9E9,9E9]],speeddata0,DefaultBlend,tool0;
  MoveAbsJ [[154.89,-48.81,-149.47,-24.75,-70.87,-5.15],[9E9,9E9,9E9,9E9,9E9,9E9]],speeddata0,DefaultBlend,tool0;
  MoveAbsJ [[154.62,-48.57,-149.87,-25.74,-70.66,-4.62],[9E9,9E9,9E9,9E9,9E9,9E9]],speeddata0,DefaultBlend,tool0;
  MoveAbsJ [[154.36,-48.34,-150.28,-26.73,-70.46,-4.09],[9E9,9E9,9E9,9E9,9E9,9E9]],speeddata0,DefaultBlend,tool0;
  MoveAbsJ [[154.09,-48.10,-150.68,-27.72,-70.26,-3.56],[9E9,9E9,9E9,9E9,9E9,9E9]],speeddata0,DefaultBlend,tool0;
  MoveAbsJ [[153.82,-47.87,-151.08,-28.71,-70.06,-3.03],[9E9,9E9,9E9,9E9,9E9,9E9]],speeddata0,DefaultBlend,tool0;
  MoveAbsJ [[153.56,-47.64,-151.49,-29.70,-69.85,-2.50],[9E9,9E9,9E9,9E9,9E9,9E9]],speeddata0,DefaultBlend,tool0;
  MoveAbsJ [[153.29,-47.40,-151.89,-30.69,-69.65,-1.96],[9E9,9E9,9E9,9E9,9E9,9E9]],speeddata0,DefaultBlend,tool0;
  MoveAbsJ [[153.02,-47.17,-152.29,-31.68,-69.45,-1.43],[9E9,9E9,9E9,9E9,9E9,9E9]],speeddata0,DefaultBlend,tool0;
  MoveAbsJ [[152.75,-46.93,-152.70,-32.67,-69.24,-0.90],[9E9,9E9,9E9,9E9,9E9,9E9]],speeddata0,DefaultBlend,tool0;
  MoveAbsJ [[152.49,-46.70,-153.10,-33.66,-69.04,-0.37],[9E9,9E9,9E9,9E9,9E9,9E9]],speeddata0,DefaultBlend,tool0;
  MoveAbsJ [[152.22,-46.47,-153.50,-34.65,-68.84,0.16],[9E9,9E9,9E9,9E9,9E9,9E9]],speeddata0,DefaultBlend,tool0;
  MoveAbsJ [[151.95,-46.23,-153.90,-35.64,-68.63,0.69],[9E9,9E9,9E9,9E9,9E9,9E9]],speeddata0,DefaultBlend,tool0;
  MoveAbsJ [[151.69,-46.00,-154.31,-36.63,-68.43,1.22],[9E9,9E9,9E9,9E9,9E9,9E9]],speeddata0,DefaultBlend,tool0;
  MoveAbsJ [[151.42,-45.76,-154.71,-37.62,-68.23,1.75],[9E9,9E9,9E9,9E9,9E9,9E9]],speeddata0,DefaultBlend,tool0;
  MoveAbsJ [[151.15,-45.53,-155.11,-38.61,-68.02,2.29],[9E9,9E9,9E9,9E9,9E9,9E9]],speeddata0,DefaultBlend,tool0;
  MoveAbsJ [[150.89,-45.29,-155.52,-39.60,-67.82,2.82],[9E9,9E9,9E9,9E9,9E9,9E9]],speeddata0,DefaultBlend,tool0;
  MoveAbsJ [[150.62,-45.06,-155.92,-40.59,-67.62,3.35],[9E9,9E9,9E9,9E9,9E9,9E9]],speeddata0,DefaultBlend,tool0;
  MoveAbsJ [[150.35,-44.83,-156.32,-41.58,-67.41,3.88],[9E9,9E9,9E9,9E9,9E9,9E9]],speeddata0,DefaultBlend,tool0;
  MoveAbsJ [[150.08,-44.59,-156.73,-42.57,-67.21,4.41],[9E9,9E9,9E9,9E9,9E9,9E9]],speeddata0,DefaultBlend,tool0;
  MoveAbsJ [[149.82,-44.36,-157.13,-43.56,-67.01,4.94],[9E9,9E9,9E9,9E9,9E9,9E9]],speeddata0,DefaultBlend,tool0;
  MoveAbsJ [[149.55,-44.12,-157.53,-44.55,-66.80,5.47],[9E9,9E9,9E9,9E9,9E9,9E9]],speeddata0,DefaultBlend,tool0;
  MoveAbsJ [[149.28,-43.89,-157.94,-45.54,-66.60,6.01],[9E9,9E9,9E9,9E9,9E9,9E9]],speeddata0,DefaultBlend,tool0;
  MoveAbsJ [[149.02,-43.66,-158.34,-46.53,-66.40,6.54],[9E9,9E9,9E9,9E9,9E9,9E9]],speeddata0,DefaultBlend,tool0;
  MoveAbsJ [[148.75,-43.42,-158.74,-47.52,-66.19,7.07],[9E9,9E9,9E9,9E9,9E9,9E9]],speeddata0,DefaultBlend,tool0;
  MoveAbsJ [[148.48,-43.19,-159.15,-48.51,-65.99,7.60],[9E9,9E9,9E9,9E9,9E9,9E9]],speeddata0,DefaultBlend,tool0;
  MoveAbsJ [[148.22,-42.95,-159.55,-49.50,-65.79,8.13],[9E9,9E9,9E9,9E9,9E9,9E9]],speeddata0,DefaultBlend,tool0;
  MoveAbsJ [[147.95,-42.72,-159.95,-50.49,-65.59,8.66],[9E9,9E9,9E9,9E9,9E9,9E9]],speeddata0,DefaultBlend,tool0;
  MoveAbsJ [[147.68,-42.48,-160.35,-51.48,-65.38,9.19],[9E9,9E9,9E9,9E9,9E9,9E9]],speeddata0,DefaultBlend,tool0;
  MoveAbsJ [[147.41,-42.25,-160.76,-52.47,-65.18,9.72],[9E9,9E9,9E9,9E9,9E9,9E9]],speeddata0,DefaultBlend,tool0;
  MoveAbsJ [[147.15,-42.02,-161.16,-53.46,-64.98,10.26],[9E9,9E9,9E9,9E9,9E9,9E9]],speeddata0,DefaultBlend,tool0;
  MoveAbsJ [[146.88,-41.78,-161.56,-54.45,-64.77,10.79],[9E9,9E9,9E9,9E9,9E9,9E9]],speeddata0,DefaultBlend,tool0;
  MoveAbsJ [[146.61,-41.55,-161.97,-55.44,-64.57,11.32],[9E9,9E9,9E9,9E9,9E9,9E9]],speeddata0,DefaultBlend,tool0;
  MoveAbsJ [[146.35,-41.31,-162.37,-56.43,-64.37,11.85],[9E9,9E9,9E9,9E9,9E9,9E9]],speeddata0,DefaultBlend,tool0;
  MoveAbsJ [[146.08,-41.08,-162.77,-57.42,-64.16,12.38],[9E9,9E9,9E9,9E9,9E9,9E9]],speeddata0,DefaultBlend,tool0;
  MoveAbsJ [[145.81,-40.85,-163.18,-58.41,-63.96,12.91],[9E9,9E9,9E9,9E9,9E9,9E9]],speeddata0,DefaultBlend,tool0;
  MoveAbsJ [[145.55,-40.61,-163.58,-59.40,-63.76,13.44],[9E9,9E9,9E9,9E9,9E9,9E9]],speeddata0,DefaultBlend,tool0;
  MoveAbsJ [[145.28,-40.38,-163.98,-60.39,-63.55,13.98],[9E9,9E9,9E9,9E9,9E9,9E9]],speeddata0,DefaultBlend,tool0;
  MoveAbsJ [[145.01,-40.14,-164.39,-61.38,-63.35,14.51],[9E9,9E9,9E9,9E9,9E9,9E9]],speeddata0,DefaultBlend,tool0;
  MoveAbsJ [[144.74,-39.91,-164.79,-62.37,-63.15,15.04],[9E9,9E9,9E9,9E9,9E9,9E9]],speeddata0,DefaultBlend,tool0;
  MoveAbsJ [[144.48,-39.67,-165.19,-63.36,-62.94,15.57],[9E9,9E9,9E9,9E9,9E9,9E9]],speeddata0,DefaultBlend,tool0;
  MoveAbsJ [[144.21,-39.44,-165.60,-64.35,-62.74,16.10],[9E9,9E9,9E9,9E9,9E9,9E9]],speeddata0,DefaultBlend,tool0;
  MoveAbsJ [[143.94,-39.21,-166.00,-65.34,-62.54,16.63],[9E9,9E9,9E9,9E9,9E9,9E9]],speeddata0,DefaultBlend,tool0;
  MoveAbsJ [[143.68,-38.97,-166.40,-66.33,-62.33,17.16],[9E9,9E9,9E9,9E9,9E9,9E9]],speeddata0,DefaultBlend,tool0;
  MoveAbsJ [[143.41,-38.74,-166.80,-67.32,-62.13,17.69],[9E9,9E9,9E9,9E9,9E9,9E9]],speeddata0,DefaultBlend,tool0;
  MoveAbsJ [[143.14,-38.50,-167.21,-68.31,-61.93,18.23],[9E9,9E9,9E9,9E9,9E9,9E9]],speeddata0,DefaultBlend,tool0;
  MoveAbsJ [[142.88,-38.27,-167.61,-69.30,-61.72,18.76],[9E9,9E9,9E9,9E9,9E9,9E9]],speeddata0,DefaultBlend,tool0;
  MoveAbsJ [[142.61,-38.04,-168.01,-70.29,-61.52,19.29],[9E9,9E9,9E9,9E9,9E9,9E9]],speeddata0,DefaultBlend,tool0;
  MoveAbsJ [[142.34,-37.80,-168.42,-71.28,-61.32,19.82],[9E9,9E9,9E9,9E9,9E9,9E9]],speeddata0,DefaultBlend,tool0;
  MoveAbsJ [[142.07,-37.57,-168.82,-72.27,-61.12,20.35],[9E9,9E9,9E9,9E9,9E9,9E9]],speeddata0,DefaultBlend,tool0;
  MoveAbsJ [[141.81,-37.33,-169.22,-73.26,-60.91,20.88],[9E9,9E9,9E9,9E9,9E9,9E9]],speeddata0,DefaultBlend,tool0;
  MoveAbsJ [[141.54,-37.10,-169.63,-74.25,-60.71,21.41],[9E9,9E9,9E9,9E9,9E9,9E9]],speeddata0,DefaultBlend,tool0;
  MoveAbsJ [[141.27,-36.87,-170.03,-75.24,-60.51,21.94],[9E9,9E9,9E9,9E9,9E9,9E9]],speeddata0,DefaultBlend,tool0;
  MoveAbsJ [[141.01,-36.63,-170.43,-76.23,-60.30,22.48],[9E9,9E9,9E9,9E9,9E9,9E9]],speeddata0,DefaultBlend,tool0;
  MoveAbsJ [[140.74,-36.40,-170.84,-77.22,-60.10,23.01],[9E9,9E9,9E9,9E9,9E9,9E9]],speeddata0,DefaultBlend,tool0;
  MoveAbsJ [[140.47,-36.16,-171.24,-78.21,-59.90,23.54],[9E9,9E9,9E9,9E9,9E9,9E9]],speeddata0,DefaultBlend,tool0;
  MoveAbsJ [[140.21,-35.93,-171.64,-79.19,-59.69,24.07],[9E9,9E9,9E9,9E9,9E9,9E9]],speeddata0,DefaultBlend,tool0;
  MoveAbsJ [[139.94,-35.69,-172.05,-80.18,-59.49,24.60],[9E9,9E9,9E9,9E9,9E9,9E9]],speeddata0,DefaultBlend,tool0;
  MoveAbsJ [[139.67,-35.46,-172.45,-81.17,-59.29,25.13],[9E9,9E9,9E9,9E9,9E9,9E9]],speeddata0,DefaultBlend,tool0;
  MoveAbsJ [[139.40,-35.23,-172.85,-82.16,-59.08,25.66],[9E9,9E9,9E9,9E9,9E9,9E9]],speeddata0,DefaultBlend,tool0;
  MoveAbsJ [[139.14,-34.99,-173.26,-83.15,-58.88,26.20],[9E9,9E9,9E9,9E9,9E9,9E9]],speeddata0,DefaultBlend,tool0;
  MoveAbsJ [[138.87,-34.76,-173.66,-84.14,-58.68,26.73],[9E9,9E9,9E9,9E9,9E9,9E9]],speeddata0,DefaultBlend,tool0;
  MoveAbsJ [[138.60,-34.52,-174.06,-85.13,-58.47,27.26],[9E9,9E9,9E9,9E9,9E9,9E9]],speeddata0,DefaultBlend,tool0;
  MoveAbsJ [[138.34,-34.29,-174.46,-86.12,-58.27,27.79],[9E9,9E9,9E9,9E9,9E9,9E9]],speeddata0,DefaultBlend,tool0;
  MoveAbsJ [[138.07,-34.06,-174.87,-87.11,-58.07,28.32],[9E9,9E9,9E9,9E9,9E9,9E9]],speeddata0,DefaultBlend,tool0;
  MoveAbsJ [[137.80,-33.82,-175.27,-88.10,-57.86,28.85],[9E9,9E9,9E9,9E9,9E9,9E9]],speeddata0,DefaultBlend,tool0;
  MoveAbsJ [[137.54,-33.59,-175.67,-89.09,-57.66,29.38],[9E9,9E9,9E9,9E9,9E9,9E9]],speeddata0,DefaultBlend,tool0;
  MoveAbsJ [[137.27,-33.35,-176.08,-90.08,-57.46,29.91],[9E9,9E9,9E9,9E9,9E9,9E9]],speeddata0,DefaultBlend,tool0;
  MoveAbsJ [[137.00,-33.12,-176.48,-91.07,-57.25,30.45],[9E9,9E9,9E9,9E9,9E9,9E9]],speeddata0,DefaultBlend,tool0;
  MoveAbsJ [[136.73,-32.88,-176.88,-92.06,-57.05,30.98],[9E9,9E9,9E9,9E9,9E9,9E9]],speeddata0,DefaultBlend,tool0;
  MoveAbsJ [[136.47,-32.65,-177.29,-93.05,-56.85,31.51],[9E9,9E9,9E9,9E9,9E9,9E9]],speeddata0,DefaultBlend,tool0;
  MoveAbsJ [[136.20,-32.42,-177.69,-94.04,-56.65,32.04],[9E9,9E9,9E9,9E9,9E9,9E9]],speeddata0,DefaultBlend,tool0;
  MoveAbsJ [[135.93,-32.18,-178.09,-95.03,-56.44,32.57],[9E9,9E9,9E9,9E9,9E9,9E9]],speeddata0,DefaultBlend,tool0;
  MoveAbsJ [[135.67,-31.95,-178.50,-96.02,-56.24,33.10],[9E9,9E9,9E9,9E9,9E9,9E9]],speeddata0,DefaultBlend,tool0;
  MoveAbsJ [[135.40,-31.71,-178.90,-97.01,-56.04,33.63],[9E9,9E9,9E9,9E9,9E9,9E9]],speeddata0,DefaultBlend,tool0;
  MoveAbsJ [[135.13,-31.48,-179.30,-98.00,-55.83,34.17],[9E9,9E9,9E9,9E9,9E9,9E9]],speeddata0,DefaultBlend,tool0;
  MoveAbsJ [[134.87,-31.25,-179.71,-98.99,-55.63,34.70],[9E9,9E9,9E9,9E9,9E9,9E9]],speeddata0,DefaultBlend,tool0;
  MoveAbsJ [[134.60,-31.01,-180.11,-99.98,-55.43,35.23],[9E9,9E9,9E9,9E9,9E9,9E9]],speeddata0,DefaultBlend,tool0;
  MoveAbsJ [[134.33,-30.78,-180.51,-100.97,-55.22,35.76],[9E9,9E9,9E9,9E9,9E9,9E9]],speeddata0,DefaultBlend,tool0;
  MoveAbsJ [[134.06,-30.54,-180.91,-101.96,-55.02,36.29],[9E9,9E9,9E9,9E9,9E9,9E9]],speeddata0,DefaultBlend,tool0;
  MoveAbsJ [[133.80,-30.31,-181.32,-102.95,-54.82,36.82],[9E9,9E9,9E9,9E9,9E9,9E9]],speeddata0,DefaultBlend,tool0;
  MoveAbsJ [[133.53,-30.07,-181.72,-103.94,-54.61,37.35],[9E9,9E9,9E9,9E9,9E9,9E9]],speeddata0,DefaultBlend,tool0;
  MoveAbsJ [[133.26,-29.84,-182.12,-104.93,-54.41,37.88],[9E9,9E9,9E9,9E9,9E9,9E9]],speeddata0,DefaultBlend,tool0;
  MoveAbsJ [[133.00,-29.61,-182.53,-105.92,-54.21,38.42],[9E9,9E9,9E9,9E9,9E9,9E9]],speeddata0,DefaultBlend,tool0;
  MoveAbsJ [[132.73,-29.37,-182.93,-106.91,-54.00,38.95],[9E9,9E9,9E9,9E9,9E9,9E9]],speeddata0,DefaultBlend,tool0;
  MoveAbsJ [[132.46,-29.14,-183.33,-107.90,-53.80,39.48],[9E9,9E9,9E9,9E9,9E9,9E9]],speeddata0,DefaultBlend,tool0;
  MoveAbsJ [[132.20,-28.90,-183.74,-108.89,-53.60,40.01],[9E9,9E9,9E9,9E9,9E9,9E9]],speeddata0,DefaultBlend,tool0;
  MoveAbsJ [[131.93,-28.67,-184.14,-109.88,-53.39,40.54],[9E9,9E9,9E9,9E9,9E9,9E9]],speeddata0,DefaultBlend,tool0;
  MoveAbsJ [[131.66,-28.44,-184.54,-110.87,-53.19,41.07],[9E9,9E9,9E9,9E9,9E9,9E9]],speeddata0,DefaultBlend,tool0;
  MoveAbsJ [[131.39,-28.20,-184.95,-111.86,-52.99,41.60],[9E9,9E9,9E9,9E9,9E9,9E9]],speeddata0,DefaultBlend,tool0;
  MoveAbsJ [[131.13,-27.97,-185.35,-112.85,-52.78,42.13],[9E9,9E9,9E9,9E9,9E9,9E9]],speeddata0,DefaultBlend,tool0;
  MoveAbsJ [[130.86,-27.73,-185.75,-113.84,-52.58,42.67],[9E9,9E9,9E9,9E9,9E9,9E9]],speeddata0,DefaultBlend,tool0;
  MoveAbsJ [[130.59,-27.50,-186.16,-114.83,-52.38,43.20],[9E9,9E9,9E9,9E9,9E9,9E9]],speeddata0,DefaultBlend,tool0;
  MoveAbsJ [[130.33,-27.27,-186.56,-115.82,-52.18,43.73],[9E9,9E9,9E9,9E9,9E9,9E9]],speeddata0,DefaultBlend,tool0;
  MoveAbsJ [[130.06,-27.03,-186.96,-116.81,-51.97,44.26],[9E9,9E9,9E9,9E9,9E9,9E9]],speeddata0,DefaultBlend,tool0;
  MoveAbsJ [[129.79,-26.80,-187.36,-117.80,-51.77,44.79],[9E9,9E9,9E9,9E9,9E9,9E9]],speeddata0,DefaultBlend,tool0;
  MoveAbsJ [[129.53,-26.56,-187.77,-118.79,-51.57,45.32],[9E9,9E9,9E9,9E9,9E9,9E9]],speeddata0,DefaultBlend,tool0;
  MoveAbsJ [[129.26,-26.33,-188.17,-119.78,-51.36,45.85],[9E9,9E9,9E9,9E9,9E9,9E9]],speeddata0,DefaultBlend,tool0;
  MoveAbsJ [[128.99,-26.09,-188.57,-120.77,-51.16,46.39],[9E9,9E9,9E9,9E9,9E9,9E9]],speeddata0,DefaultBlend,tool0;
  MoveAbsJ [[128.73,-25.86,-188.98,-121.76,-50.96,46.92],[9E9,9E9,9E9,9E9,9E9,9E9]],speeddata0,DefaultBlend,tool0;
  MoveAbsJ [[128.46,-25.63,-189.38,-122.75,-50.75,47.45],[9E9,9E9,9E9,9E9,9E9,9E9]],speeddata0,DefaultBlend,tool0;
  MoveAbsJ [[128.19,-25.39,-189.78,-123.74,-50.55,47.98],[9E9,9E9,9E9,9E9,9E9,9E9]],speeddata0,DefaultBlend,tool0;
  MoveAbsJ [[127.92,-25.16,-190.19,-124.73,-50.35,48.51],[9E9,9E9,9E9,9E9,9E9,9E9]],speeddata0,DefaultBlend,tool0;
  MoveAbsJ [[127.66,-24.92,-190.59,-125.72,-50.14,49.04],[9E9,9E9,9E9,9E9,9E9,9E9]],speeddata0,DefaultBlend,tool0;
  MoveAbsJ [[127.39,-24.69,-190.99,-126.71,-49.94,49.57],[9E9,9E9,9E9,9E9,9E9,9E9]],speeddata0,DefaultBlend,tool0;
  MoveAbsJ [[127.12,-24.46,-191.40,-127.70,-49.74,50.10],[9E9,9E9,9E9,9E9,9E9,9E9]],speeddata0,FinePoint,tool0;
  TPWrite "Action 15 LoadWorkpiece.";
  TPWrite "Press Play to Continue";
  Stop;
  TPWrite "Action 16 CloseGripper.";
  TPWrite "Press Play to Continue";
  Stop;
  TPWrite "Action 17 FreeMovement.";
  MoveAbsJ [[127.12,-24.46,-191.40,-127.70,-49.74,50.10],[9E9,9E9,9E9,9E9,9E9,9E9]],speeddata0,DefaultBlend,tool0;
  MoveAbsJ [[127.53,-24.54,-191.20,-126.71,-49.88,50.41],[9E9,9E9,9E9,9E9,9E9,9E9]],speeddata0,DefaultBlend,tool0;
  MoveAbsJ [[127.94,-24.63,-191.00,-125.72,-50.03,50.72],[9E9,9E9,9E9,9E9,9E9,9E9]],speeddata0,DefaultBlend,tool0;
  MoveAbsJ [[128.35,-24.72,-190.80,-124.73,-50.17,51.03],[9E9,9E9,9E9,9E9,9E9,9E9]],speeddata0,DefaultBlend,tool0;
  MoveAbsJ [[128.76,-24.80,-190.60,-123.74,-50.32,51.34],[9E9,9E9,9E9,9E9,9E9,9E9]],speeddata0,DefaultBlend,tool0;
  MoveAbsJ [[129.17,-24.89,-190.41,-122.75,-50.46,51.65],[9E9,9E9,9E9,9E9,9E9,9E9]],speeddata0,DefaultBlend,tool0;
  MoveAbsJ [[129.58,-24.98,-190.21,-121.76,-50.61,51.96],[9E9,9E9,9E9,9E9,9E9,9E9]],speeddata0,DefaultBlend,tool0;
  MoveAbsJ [[129.99,-25.06,-190.01,-120.77,-50.75,52.27],[9E9,9E9,9E9,9E9,9E9,9E9]],speeddata0,DefaultBlend,tool0;
  MoveAbsJ [[130.40,-25.15,-189.81,-119.78,-50.90,52.58],[9E9,9E9,9E9,9E9,9E9,9E9]],speeddata0,DefaultBlend,tool0;
  MoveAbsJ [[130.81,-25.24,-189.61,-118.79,-51.05,52.89],[9E9,9E9,9E9,9E9,9E9,9E9]],speeddata0,DefaultBlend,tool0;
  MoveAbsJ [[131.22,-25.32,-189.42,-117.80,-51.19,53.20],[9E9,9E9,9E9,9E9,9E9,9E9]],speeddata0,DefaultBlend,tool0;
  MoveAbsJ [[131.63,-25.41,-189.22,-116.81,-51.34,53.51],[9E9,9E9,9E9,9E9,9E9,9E9]],speeddata0,DefaultBlend,tool0;
  MoveAbsJ [[132.04,-25.50,-189.02,-115.82,-51.48,53.82],[9E9,9E9,9E9,9E9,9E9,9E9]],speeddata0,DefaultBlend,tool0;
  MoveAbsJ [[132.45,-25.58,-188.82,-114.83,-51.63,54.12],[9E9,9E9,9E9,9E9,9E9,9E9]],speeddata0,DefaultBlend,tool0;
  MoveAbsJ [[132.86,-25.67,-188.63,-113.84,-51.77,54.43],[9E9,9E9,9E9,9E9,9E9,9E9]],speeddata0,DefaultBlend,tool0;
  MoveAbsJ [[133.27,-25.76,-188.43,-112.85,-51.92,54.74],[9E9,9E9,9E9,9E9,9E9,9E9]],speeddata0,DefaultBlend,tool0;
  MoveAbsJ [[133.68,-25.84,-188.23,-111.86,-52.06,55.05],[9E9,9E9,9E9,9E9,9E9,9E9]],speeddata0,DefaultBlend,tool0;
  MoveAbsJ [[134.09,-25.93,-188.03,-110.87,-52.21,55.36],[9E9,9E9,9E9,9E9,9E9,9E9]],speeddata0,DefaultBlend,tool0;
  MoveAbsJ [[134.50,-26.02,-187.83,-109.88,-52.35,55.67],[9E9,9E9,9E9,9E9,9E9,9E9]],speeddata0,DefaultBlend,tool0;
  MoveAbsJ [[134.91,-26.10,-187.64,-108.89,-52.50,55.98],[9E9,9E9,9E9,9E9,9E9,9E9]],speeddata0,DefaultBlend,tool0;
  MoveAbsJ [[135.32,-26.19,-187.44,-107.90,-52.64,56.29],[9E9,9E9,9E9,9E9,9E9,9E9]],speeddata0,DefaultBlend,tool0;
